KUKA KRL program: draw2.src

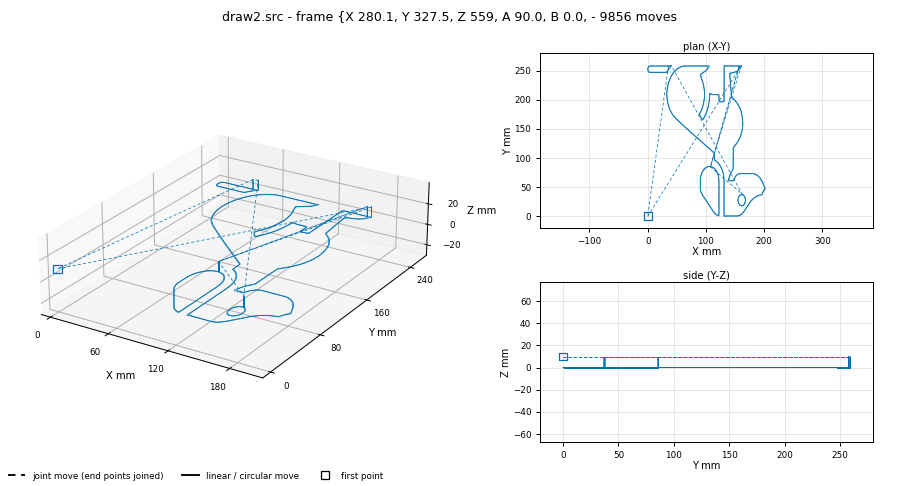
[picture p0: tool path of draw2.src in frame {X 280.1, Y 327.5, Z 559, A 90.0, B 0.0,, 9856 of 9857 moves have a stored position in this frame; points joined in program order, loops and branches not executed]
&ACCESS RVP
&REL 1
DEF DRAW_PICTURE()
; Define home position (pencil up)
POS p_home
p_home = {X 0.00, Y 0.00, Z 10.00, A 0, B 0, C 0}

BAS(#initmov, 0)

$TOOL={X -139.8, Y -0.9, Z 136.2, A 0.0, B 180.0, C 0.0}
$BASE={X 280.1, Y 327.5, Z 559, A 90.0, B 0.0, C 0.0}

PTP $axis_act

PTP p_home

; ----- Contour 1 -----
PTP {X 160.54, Y 258.89, Z 10.00, A 0, B 0, C 0}
LIN {X 160.54, Y 258.89, Z 0.00, A 0, B 0, C 0}
LIN {X 160.34, Y 258.73, Z 0.00, A 0, B 0, C 0} C_DIS
LIN {X 160.14, Y 258.62, Z 0.00, A 0, B 0, C 0} C_DIS
LIN {X 159.93, Y 258.53, Z 0.00, A 0, B 0, C 0} C_DIS
LIN {X 159.72, Y 258.48, Z 0.00, A 0, B 0, C 0} C_DIS
LIN {X 159.50, Y 258.44, Z 0.00, A 0, B 0, C 0} C_DIS
LIN {X 159.29, Y 258.42, Z 0.00, A 0, B 0, C 0} C_DIS
LIN {X 159.07, Y 258.41, Z 0.00, A 0, B 0, C 0} C_DIS
LIN {X 158.85, Y 258.41, Z 0.00, A 0, B 0, C 0} C_DIS
LIN {X 158.63, Y 258.40, Z 0.00, A 0, B 0, C 0} C_DIS
LIN {X 158.41, Y 258.40, Z 0.00, A 0, B 0, C 0} C_DIS
LIN {X 158.20, Y 258.40, Z 0.00, A 0, B 0, C 0} C_DIS
LIN {X 157.98, Y 258.40, Z 0.00, A 0, B 0, C 0} C_DIS
LIN {X 157.76, Y 258.40, Z 0.00, A 0, B 0, C 0} C_DIS
LIN {X 157.54, Y 258.40, Z 0.00, A 0, B 0, C 0} C_DIS
LIN {X 157.33, Y 258.40, Z 0.00, A 0, B 0, C 0} C_DIS
LIN {X 157.11, Y 258.40, Z 0.00, A 0, B 0, C 0} C_DIS
LIN {X 156.89, Y 258.41, Z 0.00, A 0, B 0, C 0} C_DIS
LIN {X 156.67, Y 258.41, Z 0.00, A 0, B 0, C 0} C_DIS
LIN {X 156.46, Y 258.41, Z 0.00, A 0, B 0, C 0} C_DIS
LIN {X 156.24, Y 258.41, Z 0.00, A 0, B 0, C 0} C_DIS
LIN {X 156.02, Y 258.41, Z 0.00, A 0, B 0, C 0} C_DIS
LIN {X 155.81, Y 258.41, Z 0.00, A 0, B 0, C 0} C_DIS
LIN {X 155.59, Y 258.41, Z 0.00, A 0, B 0, C 0} C_DIS
LIN {X 155.37, Y 258.41, Z 0.00, A 0, B 0, C 0} C_DIS
LIN {X 155.15, Y 258.41, Z 0.00, A 0, B 0, C 0} C_DIS
LIN {X 154.94, Y 258.41, Z 0.00, A 0, B 0, C 0} C_DIS
LIN {X 154.72, Y 258.41, Z 0.00, A 0, B 0, C 0} C_DIS
LIN {X 154.50, Y 258.41, Z 0.00, A 0, B 0, C 0} C_DIS
LIN {X 154.28, Y 258.41, Z 0.00, A 0, B 0, C 0} C_DIS
LIN {X 154.07, Y 258.41, Z 0.00, A 0, B 0, C 0} C_DIS
LIN {X 153.85, Y 258.41, Z 0.00, A 0, B 0, C 0} C_DIS
LIN {X 153.63, Y 258.41, Z 0.00, A 0, B 0, C 0} C_DIS
LIN {X 153.41, Y 258.41, Z 0.00, A 0, B 0, C 0} C_DIS
LIN {X 153.20, Y 258.41, Z 0.00, A 0, B 0, C 0} C_DIS
LIN {X 152.98, Y 258.41, Z 0.00, A 0, B 0, C 0} C_DIS
LIN {X 152.76, Y 258.41, Z 0.00, A 0, B 0, C 0} C_DIS
LIN {X 152.54, Y 258.41, Z 0.00, A 0, B 0, C 0} C_DIS
LIN {X 152.33, Y 258.41, Z 0.00, A 0, B 0, C 0} C_DIS
LIN {X 152.11, Y 258.41, Z 0.00, A 0, B 0, C 0} C_DIS
LIN {X 151.89, Y 258.41, Z 0.00, A 0, B 0, C 0} C_DIS
LIN {X 151.67, Y 258.41, Z 0.00, A 0, B 0, C 0} C_DIS
LIN {X 151.46, Y 258.41, Z 0.00, A 0, B 0, C 0} C_DIS
LIN {X 151.24, Y 258.41, Z 0.00, A 0, B 0, C 0} C_DIS
LIN {X 151.02, Y 258.41, Z 0.00, A 0, B 0, C 0} C_DIS
LIN {X 150.80, Y 258.41, Z 0.00, A 0, B 0, C 0} C_DIS
LIN {X 150.59, Y 258.41, Z 0.00, A 0, B 0, C 0} C_DIS
LIN {X 150.37, Y 258.41, Z 0.00, A 0, B 0, C 0} C_DIS
LIN {X 150.15, Y 258.41, Z 0.00, A 0, B 0, C 0} C_DIS
LIN {X 149.93, Y 258.41, Z 0.00, A 0, B 0, C 0} C_DIS
LIN {X 149.72, Y 258.41, Z 0.00, A 0, B 0, C 0} C_DIS
LIN {X 149.50, Y 258.41, Z 0.00, A 0, B 0, C 0} C_DIS
LIN {X 149.28, Y 258.41, Z 0.00, A 0, B 0, C 0} C_DIS
LIN {X 149.06, Y 258.41, Z 0.00, A 0, B 0, C 0} C_DIS
LIN {X 148.85, Y 258.41, Z 0.00, A 0, B 0, C 0} C_DIS
LIN {X 148.63, Y 258.41, Z 0.00, A 0, B 0, C 0} C_DIS
LIN {X 148.41, Y 258.41, Z 0.00, A 0, B 0, C 0} C_DIS
LIN {X 148.19, Y 258.41, Z 0.00, A 0, B 0, C 0} C_DIS
LIN {X 147.98, Y 258.41, Z 0.00, A 0, B 0, C 0} C_DIS
LIN {X 147.76, Y 258.41, Z 0.00, A 0, B 0, C 0} C_DIS
LIN {X 147.54, Y 258.41, Z 0.00, A 0, B 0, C 0} C_DIS
LIN {X 147.33, Y 258.41, Z 0.00, A 0, B 0, C 0} C_DIS
LIN {X 147.11, Y 258.41, Z 0.00, A 0, B 0, C 0} C_DIS
LIN {X 146.89, Y 258.41, Z 0.00, A 0, B 0, C 0} C_DIS
LIN {X 146.67, Y 258.41, Z 0.00, A 0, B 0, C 0} C_DIS
LIN {X 146.46, Y 258.41, Z 0.00, A 0, B 0, C 0} C_DIS
LIN {X 146.24, Y 258.41, Z 0.00, A 0, B 0, C 0} C_DIS
LIN {X 146.02, Y 258.41, Z 0.00, A 0, B 0, C 0} C_DIS
LIN {X 145.80, Y 258.41, Z 0.00, A 0, B 0, C 0} C_DIS
LIN {X 145.59, Y 258.41, Z 0.00, A 0, B 0, C 0} C_DIS
LIN {X 145.37, Y 258.41, Z 0.00, A 0, B 0, C 0} C_DIS
LIN {X 145.15, Y 258.41, Z 0.00, A 0, B 0, C 0} C_DIS
LIN {X 144.93, Y 258.41, Z 0.00, A 0, B 0, C 0} C_DIS
LIN {X 144.72, Y 258.41, Z 0.00, A 0, B 0, C 0} C_DIS
LIN {X 144.50, Y 258.41, Z 0.00, A 0, B 0, C 0} C_DIS
LIN {X 144.28, Y 258.41, Z 0.00, A 0, B 0, C 0} C_DIS
LIN {X 144.06, Y 258.41, Z 0.00, A 0, B 0, C 0} C_DIS
LIN {X 143.85, Y 258.41, Z 0.00, A 0, B 0, C 0} C_DIS
LIN {X 143.63, Y 258.41, Z 0.00, A 0, B 0, C 0} C_DIS
LIN {X 143.41, Y 258.41, Z 0.00, A 0, B 0, C 0} C_DIS
LIN {X 143.19, Y 258.41, Z 0.00, A 0, B 0, C 0} C_DIS
LIN {X 142.98, Y 258.41, Z 0.00, A 0, B 0, C 0} C_DIS
LIN {X 142.76, Y 258.41, Z 0.00, A 0, B 0, C 0} C_DIS
LIN {X 142.54, Y 258.41, Z 0.00, A 0, B 0, C 0} C_DIS
LIN {X 142.32, Y 258.41, Z 0.00, A 0, B 0, C 0} C_DIS
LIN {X 142.11, Y 258.41, Z 0.00, A 0, B 0, C 0} C_DIS
LIN {X 141.89, Y 258.41, Z 0.00, A 0, B 0, C 0} C_DIS
LIN {X 141.67, Y 258.41, Z 0.00, A 0, B 0, C 0} C_DIS
LIN {X 141.45, Y 258.41, Z 0.00, A 0, B 0, C 0} C_DIS
LIN {X 141.24, Y 258.41, Z 0.00, A 0, B 0, C 0} C_DIS
LIN {X 141.02, Y 258.41, Z 0.00, A 0, B 0, C 0} C_DIS
LIN {X 140.80, Y 258.41, Z 0.00, A 0, B 0, C 0} C_DIS
LIN {X 140.58, Y 258.41, Z 0.00, A 0, B 0, C 0} C_DIS
LIN {X 140.37, Y 258.41, Z 0.00, A 0, B 0, C 0} C_DIS
LIN {X 140.15, Y 258.41, Z 0.00, A 0, B 0, C 0} C_DIS
LIN {X 139.93, Y 258.41, Z 0.00, A 0, B 0, C 0} C_DIS
LIN {X 139.71, Y 258.41, Z 0.00, A 0, B 0, C 0} C_DIS
LIN {X 139.50, Y 258.41, Z 0.00, A 0, B 0, C 0} C_DIS
LIN {X 139.28, Y 258.41, Z 0.00, A 0, B 0, C 0} C_DIS
LIN {X 139.06, Y 258.41, Z 0.00, A 0, B 0, C 0} C_DIS
LIN {X 138.85, Y 258.41, Z 0.00, A 0, B 0, C 0} C_DIS
LIN {X 138.63, Y 258.41, Z 0.00, A 0, B 0, C 0} C_DIS
LIN {X 138.41, Y 258.41, Z 0.00, A 0, B 0, C 0} C_DIS
LIN {X 138.19, Y 258.41, Z 0.00, A 0, B 0, C 0} C_DIS
LIN {X 137.98, Y 258.41, Z 0.00, A 0, B 0, C 0} C_DIS
LIN {X 137.76, Y 258.41, Z 0.00, A 0, B 0, C 0} C_DIS
LIN {X 137.54, Y 258.40, Z 0.00, A 0, B 0, C 0} C_DIS
LIN {X 137.32, Y 258.40, Z 0.00, A 0, B 0, C 0} C_DIS
LIN {X 137.11, Y 258.40, Z 0.00, A 0, B 0, C 0} C_DIS
LIN {X 136.89, Y 258.40, Z 0.00, A 0, B 0, C 0} C_DIS
LIN {X 136.67, Y 258.40, Z 0.00, A 0, B 0, C 0} C_DIS
LIN {X 136.45, Y 258.40, Z 0.00, A 0, B 0, C 0} C_DIS
LIN {X 136.24, Y 258.40, Z 0.00, A 0, B 0, C 0} C_DIS
LIN {X 136.02, Y 258.40, Z 0.00, A 0, B 0, C 0} C_DIS
LIN {X 135.80, Y 258.41, Z 0.00, A 0, B 0, C 0} C_DIS
LIN {X 135.58, Y 258.41, Z 0.00, A 0, B 0, C 0} C_DIS
LIN {X 135.37, Y 258.41, Z 0.00, A 0, B 0, C 0} C_DIS
LIN {X 135.15, Y 258.41, Z 0.00, A 0, B 0, C 0} C_DIS
LIN {X 134.93, Y 258.41, Z 0.00, A 0, B 0, C 0} C_DIS
LIN {X 134.72, Y 258.41, Z 0.00, A 0, B 0, C 0} C_DIS
LIN {X 134.50, Y 258.41, Z 0.00, A 0, B 0, C 0} C_DIS
LIN {X 134.28, Y 258.41, Z 0.00, A 0, B 0, C 0} C_DIS
LIN {X 134.06, Y 258.41, Z 0.00, A 0, B 0, C 0} C_DIS
LIN {X 133.84, Y 258.41, Z 0.00, A 0, B 0, C 0} C_DIS
LIN {X 133.63, Y 258.40, Z 0.00, A 0, B 0, C 0} C_DIS
LIN {X 133.41, Y 258.40, Z 0.00, A 0, B 0, C 0} C_DIS
LIN {X 133.19, Y 258.39, Z 0.00, A 0, B 0, C 0} C_DIS
LIN {X 132.97, Y 258.39, Z 0.00, A 0, B 0, C 0} C_DIS
LIN {X 132.75, Y 258.39, Z 0.00, A 0, B 0, C 0} C_DIS
LIN {X 132.54, Y 258.41, Z 0.00, A 0, B 0, C 0} C_DIS
LIN {X 132.32, Y 258.43, Z 0.00, A 0, B 0, C 0} C_DIS
LIN {X 132.11, Y 258.47, Z 0.00, A 0, B 0, C 0} C_DIS
LIN {X 131.90, Y 258.53, Z 0.00, A 0, B 0, C 0} C_DIS
LIN {X 131.69, Y 258.59, Z 0.00, A 0, B 0, C 0} C_DIS
LIN {X 131.47, Y 258.66, Z 0.00, A 0, B 0, C 0} C_DIS
LIN {X 131.25, Y 258.71, Z 0.00, A 0, B 0, C 0} C_DIS
LIN {X 131.03, Y 258.70, Z 0.00, A 0, B 0, C 0} C_DIS
LIN {X 130.84, Y 258.58, Z 0.00, A 0, B 0, C 0} C_DIS
LIN {X 130.73, Y 258.32, Z 0.00, A 0, B 0, C 0} C_DIS
LIN {X 130.70, Y 257.99, Z 0.00, A 0, B 0, C 0} C_DIS
LIN {X 130.73, Y 257.65, Z 0.00, A 0, B 0, C 0} C_DIS
LIN {X 130.77, Y 257.33, Z 0.00, A 0, B 0, C 0} C_DIS
LIN {X 130.83, Y 257.01, Z 0.00, A 0, B 0, C 0} C_DIS
LIN {X 130.87, Y 256.70, Z 0.00, A 0, B 0, C 0} C_DIS
LIN {X 130.90, Y 256.37, Z 0.00, A 0, B 0, C 0} C_DIS
LIN {X 130.91, Y 256.05, Z 0.00, A 0, B 0, C 0} C_DIS
LIN {X 130.91, Y 255.72, Z 0.00, A 0, B 0, C 0} C_DIS
LIN {X 130.91, Y 255.39, Z 0.00, A 0, B 0, C 0} C_DIS
LIN {X 130.91, Y 255.06, Z 0.00, A 0, B 0, C 0} C_DIS
LIN {X 130.91, Y 254.73, Z 0.00, A 0, B 0, C 0} C_DIS
LIN {X 130.91, Y 254.40, Z 0.00, A 0, B 0, C 0} C_DIS
LIN {X 130.91, Y 254.08, Z 0.00, A 0, B 0, C 0} C_DIS
LIN {X 130.91, Y 253.75, Z 0.00, A 0, B 0, C 0} C_DIS
LIN {X 130.91, Y 253.42, Z 0.00, A 0, B 0, C 0} C_DIS
LIN {X 130.91, Y 253.10, Z 0.00, A 0, B 0, C 0} C_DIS
LIN {X 130.91, Y 252.77, Z 0.00, A 0, B 0, C 0} C_DIS
LIN {X 130.91, Y 252.44, Z 0.00, A 0, B 0, C 0} C_DIS
LIN {X 130.91, Y 252.11, Z 0.00, A 0, B 0, C 0} C_DIS
LIN {X 130.91, Y 251.78, Z 0.00, A 0, B 0, C 0} C_DIS
LIN {X 130.91, Y 251.46, Z 0.00, A 0, B 0, C 0} C_DIS
LIN {X 130.91, Y 251.13, Z 0.00, A 0, B 0, C 0} C_DIS
LIN {X 130.91, Y 250.80, Z 0.00, A 0, B 0, C 0} C_DIS
LIN {X 130.91, Y 250.47, Z 0.00, A 0, B 0, C 0} C_DIS
LIN {X 130.91, Y 250.15, Z 0.00, A 0, B 0, C 0} C_DIS
LIN {X 130.91, Y 249.82, Z 0.00, A 0, B 0, C 0} C_DIS
LIN {X 130.91, Y 249.49, Z 0.00, A 0, B 0, C 0} C_DIS
LIN {X 130.91, Y 249.16, Z 0.00, A 0, B 0, C 0} C_DIS
LIN {X 130.91, Y 248.84, Z 0.00, A 0, B 0, C 0} C_DIS
LIN {X 130.91, Y 248.51, Z 0.00, A 0, B 0, C 0} C_DIS
LIN {X 130.91, Y 248.18, Z 0.00, A 0, B 0, C 0} C_DIS
LIN {X 130.91, Y 247.85, Z 0.00, A 0, B 0, C 0} C_DIS
LIN {X 130.91, Y 247.52, Z 0.00, A 0, B 0, C 0} C_DIS
LIN {X 130.91, Y 247.20, Z 0.00, A 0, B 0, C 0} C_DIS
LIN {X 130.91, Y 246.87, Z 0.00, A 0, B 0, C 0} C_DIS
LIN {X 130.91, Y 246.54, Z 0.00, A 0, B 0, C 0} C_DIS
LIN {X 130.91, Y 246.21, Z 0.00, A 0, B 0, C 0} C_DIS
LIN {X 130.91, Y 245.89, Z 0.00, A 0, B 0, C 0} C_DIS
LIN {X 130.91, Y 245.56, Z 0.00, A 0, B 0, C 0} C_DIS
LIN {X 130.91, Y 245.23, Z 0.00, A 0, B 0, C 0} C_DIS
LIN {X 130.91, Y 244.90, Z 0.00, A 0, B 0, C 0} C_DIS
LIN {X 130.91, Y 244.58, Z 0.00, A 0, B 0, C 0} C_DIS
LIN {X 130.91, Y 244.25, Z 0.00, A 0, B 0, C 0} C_DIS
LIN {X 130.91, Y 243.92, Z 0.00, A 0, B 0, C 0} C_DIS
LIN {X 130.91, Y 243.59, Z 0.00, A 0, B 0, C 0} C_DIS
LIN {X 130.91, Y 243.26, Z 0.00, A 0, B 0, C 0} C_DIS
LIN {X 130.91, Y 242.94, Z 0.00, A 0, B 0, C 0} C_DIS
LIN {X 130.91, Y 242.61, Z 0.00, A 0, B 0, C 0} C_DIS
LIN {X 130.91, Y 242.28, Z 0.00, A 0, B 0, C 0} C_DIS
LIN {X 130.91, Y 241.95, Z 0.00, A 0, B 0, C 0} C_DIS
LIN {X 130.91, Y 241.63, Z 0.00, A 0, B 0, C 0} C_DIS
LIN {X 130.91, Y 241.30, Z 0.00, A 0, B 0, C 0} C_DIS
LIN {X 130.91, Y 240.97, Z 0.00, A 0, B 0, C 0} C_DIS
LIN {X 130.91, Y 240.64, Z 0.00, A 0, B 0, C 0} C_DIS
LIN {X 130.91, Y 240.32, Z 0.00, A 0, B 0, C 0} C_DIS
LIN {X 130.91, Y 239.99, Z 0.00, A 0, B 0, C 0} C_DIS
LIN {X 130.91, Y 239.66, Z 0.00, A 0, B 0, C 0} C_DIS
LIN {X 130.91, Y 239.33, Z 0.00, A 0, B 0, C 0} C_DIS
LIN {X 130.91, Y 239.00, Z 0.00, A 0, B 0, C 0} C_DIS
LIN {X 130.91, Y 238.68, Z 0.00, A 0, B 0, C 0} C_DIS
LIN {X 130.91, Y 238.35, Z 0.00, A 0, B 0, C 0} C_DIS
LIN {X 130.91, Y 238.02, Z 0.00, A 0, B 0, C 0} C_DIS
LIN {X 130.91, Y 237.69, Z 0.00, A 0, B 0, C 0} C_DIS
LIN {X 130.91, Y 237.37, Z 0.00, A 0, B 0, C 0} C_DIS
LIN {X 130.91, Y 237.04, Z 0.00, A 0, B 0, C 0} C_DIS
LIN {X 130.91, Y 236.71, Z 0.00, A 0, B 0, C 0} C_DIS
LIN {X 130.91, Y 236.38, Z 0.00, A 0, B 0, C 0} C_DIS
LIN {X 130.91, Y 236.06, Z 0.00, A 0, B 0, C 0} C_DIS
LIN {X 130.91, Y 235.73, Z 0.00, A 0, B 0, C 0} C_DIS
LIN {X 130.91, Y 235.40, Z 0.00, A 0, B 0, C 0} C_DIS
LIN {X 130.91, Y 235.07, Z 0.00, A 0, B 0, C 0} C_DIS
LIN {X 130.91, Y 234.74, Z 0.00, A 0, B 0, C 0} C_DIS
LIN {X 130.91, Y 234.42, Z 0.00, A 0, B 0, C 0} C_DIS
LIN {X 130.91, Y 234.09, Z 0.00, A 0, B 0, C 0} C_DIS
LIN {X 130.91, Y 233.76, Z 0.00, A 0, B 0, C 0} C_DIS
LIN {X 130.91, Y 233.43, Z 0.00, A 0, B 0, C 0} C_DIS
LIN {X 130.91, Y 233.11, Z 0.00, A 0, B 0, C 0} C_DIS
LIN {X 130.91, Y 232.78, Z 0.00, A 0, B 0, C 0} C_DIS
LIN {X 130.91, Y 232.45, Z 0.00, A 0, B 0, C 0} C_DIS
LIN {X 130.91, Y 232.12, Z 0.00, A 0, B 0, C 0} C_DIS
LIN {X 130.91, Y 231.80, Z 0.00, A 0, B 0, C 0} C_DIS
LIN {X 130.91, Y 231.47, Z 0.00, A 0, B 0, C 0} C_DIS
LIN {X 130.91, Y 231.14, Z 0.00, A 0, B 0, C 0} C_DIS
LIN {X 130.91, Y 230.81, Z 0.00, A 0, B 0, C 0} C_DIS
LIN {X 130.91, Y 230.48, Z 0.00, A 0, B 0, C 0} C_DIS
LIN {X 130.91, Y 230.16, Z 0.00, A 0, B 0, C 0} C_DIS
LIN {X 130.91, Y 229.83, Z 0.00, A 0, B 0, C 0} C_DIS
LIN {X 130.91, Y 229.50, Z 0.00, A 0, B 0, C 0} C_DIS
LIN {X 130.91, Y 229.17, Z 0.00, A 0, B 0, C 0} C_DIS
LIN {X 130.91, Y 228.85, Z 0.00, A 0, B 0, C 0} C_DIS
LIN {X 130.91, Y 228.52, Z 0.00, A 0, B 0, C 0} C_DIS
LIN {X 130.91, Y 228.19, Z 0.00, A 0, B 0, C 0} C_DIS
LIN {X 130.91, Y 227.86, Z 0.00, A 0, B 0, C 0} C_DIS
LIN {X 130.91, Y 227.54, Z 0.00, A 0, B 0, C 0} C_DIS
LIN {X 130.91, Y 227.21, Z 0.00, A 0, B 0, C 0} C_DIS
LIN {X 130.91, Y 226.88, Z 0.00, A 0, B 0, C 0} C_DIS
LIN {X 130.91, Y 226.55, Z 0.00, A 0, B 0, C 0} C_DIS
LIN {X 130.91, Y 226.22, Z 0.00, A 0, B 0, C 0} C_DIS
LIN {X 130.91, Y 225.90, Z 0.00, A 0, B 0, C 0} C_DIS
LIN {X 130.91, Y 225.57, Z 0.00, A 0, B 0, C 0} C_DIS
LIN {X 130.91, Y 225.24, Z 0.00, A 0, B 0, C 0} C_DIS
LIN {X 130.91, Y 224.91, Z 0.00, A 0, B 0, C 0} C_DIS
LIN {X 130.91, Y 224.59, Z 0.00, A 0, B 0, C 0} C_DIS
LIN {X 130.91, Y 224.26, Z 0.00, A 0, B 0, C 0} C_DIS
LIN {X 130.91, Y 223.93, Z 0.00, A 0, B 0, C 0} C_DIS
LIN {X 130.91, Y 223.60, Z 0.00, A 0, B 0, C 0} C_DIS
LIN {X 130.91, Y 223.28, Z 0.00, A 0, B 0, C 0} C_DIS
LIN {X 130.91, Y 222.95, Z 0.00, A 0, B 0, C 0} C_DIS
LIN {X 130.91, Y 222.62, Z 0.00, A 0, B 0, C 0} C_DIS
LIN {X 130.91, Y 222.29, Z 0.00, A 0, B 0, C 0} C_DIS
LIN {X 130.91, Y 221.96, Z 0.00, A 0, B 0, C 0} C_DIS
LIN {X 130.91, Y 221.64, Z 0.00, A 0, B 0, C 0} C_DIS
LIN {X 130.91, Y 221.31, Z 0.00, A 0, B 0, C 0} C_DIS
LIN {X 130.91, Y 220.98, Z 0.00, A 0, B 0, C 0} C_DIS
LIN {X 130.91, Y 220.65, Z 0.00, A 0, B 0, C 0} C_DIS
LIN {X 130.91, Y 220.33, Z 0.00, A 0, B 0, C 0} C_DIS
LIN {X 130.91, Y 220.00, Z 0.00, A 0, B 0, C 0} C_DIS
LIN {X 130.91, Y 219.67, Z 0.00, A 0, B 0, C 0} C_DIS
LIN {X 130.91, Y 219.34, Z 0.00, A 0, B 0, C 0} C_DIS
LIN {X 130.91, Y 219.02, Z 0.00, A 0, B 0, C 0} C_DIS
LIN {X 130.91, Y 218.69, Z 0.00, A 0, B 0, C 0} C_DIS
LIN {X 130.91, Y 218.36, Z 0.00, A 0, B 0, C 0} C_DIS
LIN {X 130.91, Y 218.03, Z 0.00, A 0, B 0, C 0} C_DIS
LIN {X 130.91, Y 217.70, Z 0.00, A 0, B 0, C 0} C_DIS
LIN {X 130.91, Y 217.38, Z 0.00, A 0, B 0, C 0} C_DIS
LIN {X 130.91, Y 217.05, Z 0.00, A 0, B 0, C 0} C_DIS
LIN {X 130.91, Y 216.72, Z 0.00, A 0, B 0, C 0} C_DIS
LIN {X 130.91, Y 216.39, Z 0.00, A 0, B 0, C 0} C_DIS
LIN {X 130.91, Y 216.07, Z 0.00, A 0, B 0, C 0} C_DIS
LIN {X 130.91, Y 215.74, Z 0.00, A 0, B 0, C 0} C_DIS
LIN {X 130.91, Y 215.41, Z 0.00, A 0, B 0, C 0} C_DIS
LIN {X 130.91, Y 215.08, Z 0.00, A 0, B 0, C 0} C_DIS
LIN {X 130.91, Y 214.76, Z 0.00, A 0, B 0, C 0} C_DIS
LIN {X 130.91, Y 214.43, Z 0.00, A 0, B 0, C 0} C_DIS
LIN {X 130.91, Y 214.10, Z 0.00, A 0, B 0, C 0} C_DIS
LIN {X 130.91, Y 213.77, Z 0.00, A 0, B 0, C 0} C_DIS
LIN {X 130.91, Y 213.44, Z 0.00, A 0, B 0, C 0} C_DIS
LIN {X 130.91, Y 213.12, Z 0.00, A 0, B 0, C 0} C_DIS
LIN {X 130.91, Y 212.79, Z 0.00, A 0, B 0, C 0} C_DIS
LIN {X 130.91, Y 212.46, Z 0.00, A 0, B 0, C 0} C_DIS
LIN {X 130.91, Y 212.13, Z 0.00, A 0, B 0, C 0} C_DIS
LIN {X 130.91, Y 211.81, Z 0.00, A 0, B 0, C 0} C_DIS
LIN {X 130.91, Y 211.48, Z 0.00, A 0, B 0, C 0} C_DIS
LIN {X 130.91, Y 211.15, Z 0.00, A 0, B 0, C 0} C_DIS
LIN {X 130.91, Y 210.82, Z 0.00, A 0, B 0, C 0} C_DIS
LIN {X 130.91, Y 210.50, Z 0.00, A 0, B 0, C 0} C_DIS
LIN {X 130.91, Y 210.17, Z 0.00, A 0, B 0, C 0} C_DIS
LIN {X 130.91, Y 209.84, Z 0.00, A 0, B 0, C 0} C_DIS
LIN {X 130.91, Y 209.51, Z 0.00, A 0, B 0, C 0} C_DIS
LIN {X 130.91, Y 209.18, Z 0.00, A 0, B 0, C 0} C_DIS
LIN {X 130.91, Y 208.86, Z 0.00, A 0, B 0, C 0} C_DIS
LIN {X 130.91, Y 208.53, Z 0.00, A 0, B 0, C 0} C_DIS
LIN {X 130.91, Y 208.20, Z 0.00, A 0, B 0, C 0} C_DIS
LIN {X 130.91, Y 207.87, Z 0.00, A 0, B 0, C 0} C_DIS
LIN {X 130.91, Y 207.55, Z 0.00, A 0, B 0, C 0} C_DIS
LIN {X 130.91, Y 207.22, Z 0.00, A 0, B 0, C 0} C_DIS
LIN {X 130.91, Y 206.89, Z 0.00, A 0, B 0, C 0} C_DIS
LIN {X 130.91, Y 206.56, Z 0.00, A 0, B 0, C 0} C_DIS
LIN {X 130.91, Y 206.24, Z 0.00, A 0, B 0, C 0} C_DIS
LIN {X 130.91, Y 205.91, Z 0.00, A 0, B 0, C 0} C_DIS
LIN {X 130.91, Y 205.58, Z 0.00, A 0, B 0, C 0} C_DIS
LIN {X 130.91, Y 205.25, Z 0.00, A 0, B 0, C 0} C_DIS
LIN {X 130.91, Y 204.92, Z 0.00, A 0, B 0, C 0} C_DIS
LIN {X 130.91, Y 204.60, Z 0.00, A 0, B 0, C 0} C_DIS
LIN {X 130.91, Y 204.27, Z 0.00, A 0, B 0, C 0} C_DIS
LIN {X 130.91, Y 203.94, Z 0.00, A 0, B 0, C 0} C_DIS
LIN {X 130.91, Y 203.61, Z 0.00, A 0, B 0, C 0} C_DIS
LIN {X 130.91, Y 203.29, Z 0.00, A 0, B 0, C 0} C_DIS
LIN {X 130.92, Y 202.96, Z 0.00, A 0, B 0, C 0} C_DIS
LIN {X 130.92, Y 202.63, Z 0.00, A 0, B 0, C 0} C_DIS
LIN {X 130.92, Y 202.30, Z 0.00, A 0, B 0, C 0} C_DIS
LIN {X 130.92, Y 201.98, Z 0.00, A 0, B 0, C 0} C_DIS
LIN {X 130.92, Y 201.65, Z 0.00, A 0, B 0, C 0} C_DIS
LIN {X 130.91, Y 201.32, Z 0.00, A 0, B 0, C 0} C_DIS
LIN {X 130.91, Y 200.99, Z 0.00, A 0, B 0, C 0} C_DIS
LIN {X 130.91, Y 200.67, Z 0.00, A 0, B 0, C 0} C_DIS
LIN {X 130.90, Y 200.34, Z 0.00, A 0, B 0, C 0} C_DIS
LIN {X 130.88, Y 200.01, Z 0.00, A 0, B 0, C 0} C_DIS
LIN {X 130.84, Y 199.69, Z 0.00, A 0, B 0, C 0} C_DIS
LIN {X 130.78, Y 199.38, Z 0.00, A 0, B 0, C 0} C_DIS
LIN {X 130.73, Y 199.05, Z 0.00, A 0, B 0, C 0} C_DIS
LIN {X 130.67, Y 198.74, Z 0.00, A 0, B 0, C 0} C_DIS
LIN {X 130.58, Y 198.44, Z 0.00, A 0, B 0, C 0} C_DIS
LIN {X 130.45, Y 198.19, Z 0.00, A 0, B 0, C 0} C_DIS
LIN {X 130.30, Y 197.95, Z 0.00, A 0, B 0, C 0} C_DIS
LIN {X 130.14, Y 197.71, Z 0.00, A 0, B 0, C 0} C_DIS
LIN {X 129.98, Y 197.49, Z 0.00, A 0, B 0, C 0} C_DIS
LIN {X 129.81, Y 197.30, Z 0.00, A 0, B 0, C 0} C_DIS
LIN {X 129.62, Y 197.16, Z 0.00, A 0, B 0, C 0} C_DIS
LIN {X 129.42, Y 197.05, Z 0.00, A 0, B 0, C 0} C_DIS
LIN {X 129.20, Y 196.98, Z 0.00, A 0, B 0, C 0} C_DIS
LIN {X 128.98, Y 196.91, Z 0.00, A 0, B 0, C 0} C_DIS
LIN {X 128.77, Y 196.86, Z 0.00, A 0, B 0, C 0} C_DIS
LIN {X 128.56, Y 196.82, Z 0.00, A 0, B 0, C 0} C_DIS
LIN {X 128.34, Y 196.80, Z 0.00, A 0, B 0, C 0} C_DIS
LIN {X 128.12, Y 196.78, Z 0.00, A 0, B 0, C 0} C_DIS
LIN {X 127.91, Y 196.78, Z 0.00, A 0, B 0, C 0} C_DIS
LIN {X 127.69, Y 196.78, Z 0.00, A 0, B 0, C 0} C_DIS
LIN {X 127.47, Y 196.79, Z 0.00, A 0, B 0, C 0} C_DIS
LIN {X 127.26, Y 196.79, Z 0.00, A 0, B 0, C 0} C_DIS
LIN {X 127.04, Y 196.80, Z 0.00, A 0, B 0, C 0} C_DIS
LIN {X 126.82, Y 196.81, Z 0.00, A 0, B 0, C 0} C_DIS
LIN {X 126.60, Y 196.81, Z 0.00, A 0, B 0, C 0} C_DIS
LIN {X 126.38, Y 196.80, Z 0.00, A 0, B 0, C 0} C_DIS
LIN {X 126.17, Y 196.79, Z 0.00, A 0, B 0, C 0} C_DIS
LIN {X 125.95, Y 196.79, Z 0.00, A 0, B 0, C 0} C_DIS
LIN {X 125.73, Y 196.78, Z 0.00, A 0, B 0, C 0} C_DIS
LIN {X 125.51, Y 196.78, Z 0.00, A 0, B 0, C 0} C_DIS
LIN {X 125.30, Y 196.79, Z 0.00, A 0, B 0, C 0} C_DIS
LIN {X 125.08, Y 196.80, Z 0.00, A 0, B 0, C 0} C_DIS
LIN {X 124.86, Y 196.83, Z 0.00, A 0, B 0, C 0} C_DIS
LIN {X 124.65, Y 196.87, Z 0.00, A 0, B 0, C 0} C_DIS
LIN {X 124.43, Y 196.92, Z 0.00, A 0, B 0, C 0} C_DIS
LIN {X 124.22, Y 197.00, Z 0.00, A 0, B 0, C 0} C_DIS
LIN {X 124.01, Y 197.09, Z 0.00, A 0, B 0, C 0} C_DIS
LIN {X 123.80, Y 197.19, Z 0.00, A 0, B 0, C 0} C_DIS
LIN {X 123.61, Y 197.33, Z 0.00, A 0, B 0, C 0} C_DIS
LIN {X 123.45, Y 197.54, Z 0.00, A 0, B 0, C 0} C_DIS
LIN {X 123.30, Y 197.78, Z 0.00, A 0, B 0, C 0} C_DIS
LIN {X 123.14, Y 198.01, Z 0.00, A 0, B 0, C 0} C_DIS
LIN {X 122.99, Y 198.24, Z 0.00, A 0, B 0, C 0} C_DIS
LIN {X 122.87, Y 198.51, Z 0.00, A 0, B 0, C 0} C_DIS
LIN {X 122.79, Y 198.82, Z 0.00, A 0, B 0, C 0} C_DIS
LIN {X 122.73, Y 199.13, Z 0.00, A 0, B 0, C 0} C_DIS
LIN {X 122.67, Y 199.45, Z 0.00, A 0, B 0, C 0} C_DIS
LIN {X 122.63, Y 199.77, Z 0.00, A 0, B 0, C 0} C_DIS
LIN {X 122.60, Y 200.10, Z 0.00, A 0, B 0, C 0} C_DIS
LIN {X 122.58, Y 200.42, Z 0.00, A 0, B 0, C 0} C_DIS
LIN {X 122.56, Y 200.75, Z 0.00, A 0, B 0, C 0} C_DIS
LIN {X 122.56, Y 201.07, Z 0.00, A 0, B 0, C 0} C_DIS
LIN {X 122.55, Y 201.40, Z 0.00, A 0, B 0, C 0} C_DIS
LIN {X 122.55, Y 201.73, Z 0.00, A 0, B 0, C 0} C_DIS
LIN {X 122.56, Y 202.06, Z 0.00, A 0, B 0, C 0} C_DIS
LIN {X 122.56, Y 202.39, Z 0.00, A 0, B 0, C 0} C_DIS
LIN {X 122.56, Y 202.71, Z 0.00, A 0, B 0, C 0} C_DIS
LIN {X 122.57, Y 203.04, Z 0.00, A 0, B 0, C 0} C_DIS
LIN {X 122.57, Y 203.37, Z 0.00, A 0, B 0, C 0} C_DIS
LIN {X 122.57, Y 203.70, Z 0.00, A 0, B 0, C 0} C_DIS
LIN {X 122.57, Y 204.02, Z 0.00, A 0, B 0, C 0} C_DIS
LIN {X 122.57, Y 204.35, Z 0.00, A 0, B 0, C 0} C_DIS
LIN {X 122.56, Y 204.68, Z 0.00, A 0, B 0, C 0} C_DIS
LIN {X 122.56, Y 205.01, Z 0.00, A 0, B 0, C 0} C_DIS
LIN {X 122.56, Y 205.33, Z 0.00, A 0, B 0, C 0} C_DIS
LIN {X 122.56, Y 205.66, Z 0.00, A 0, B 0, C 0} C_DIS
LIN {X 122.56, Y 205.99, Z 0.00, A 0, B 0, C 0} C_DIS
LIN {X 122.55, Y 206.32, Z 0.00, A 0, B 0, C 0} C_DIS
LIN {X 122.56, Y 206.65, Z 0.00, A 0, B 0, C 0} C_DIS
LIN {X 122.56, Y 206.97, Z 0.00, A 0, B 0, C 0} C_DIS
LIN {X 122.57, Y 207.30, Z 0.00, A 0, B 0, C 0} C_DIS
LIN {X 122.58, Y 207.63, Z 0.00, A 0, B 0, C 0} C_DIS
LIN {X 122.56, Y 207.95, Z 0.00, A 0, B 0, C 0} C_DIS
LIN {X 122.52, Y 208.28, Z 0.00, A 0, B 0, C 0} C_DIS
LIN {X 122.43, Y 208.59, Z 0.00, A 0, B 0, C 0} C_DIS
LIN {X 122.31, Y 208.87, Z 0.00, A 0, B 0, C 0} C_DIS
LIN {X 122.15, Y 209.07, Z 0.00, A 0, B 0, C 0} C_DIS
LIN {X 121.95, Y 209.17, Z 0.00, A 0, B 0, C 0} C_DIS
LIN {X 121.74, Y 209.22, Z 0.00, A 0, B 0, C 0} C_DIS
LIN {X 121.52, Y 209.24, Z 0.00, A 0, B 0, C 0} C_DIS
LIN {X 121.30, Y 209.24, Z 0.00, A 0, B 0, C 0} C_DIS
LIN {X 121.08, Y 209.25, Z 0.00, A 0, B 0, C 0} C_DIS
LIN {X 120.86, Y 209.25, Z 0.00, A 0, B 0, C 0} C_DIS
LIN {X 120.64, Y 209.25, Z 0.00, A 0, B 0, C 0} C_DIS
LIN {X 120.42, Y 209.25, Z 0.00, A 0, B 0, C 0} C_DIS
LIN {X 120.20, Y 209.25, Z 0.00, A 0, B 0, C 0} C_DIS
LIN {X 119.99, Y 209.25, Z 0.00, A 0, B 0, C 0} C_DIS
LIN {X 119.77, Y 209.25, Z 0.00, A 0, B 0, C 0} C_DIS
LIN {X 119.56, Y 209.25, Z 0.00, A 0, B 0, C 0} C_DIS
LIN {X 119.34, Y 209.25, Z 0.00, A 0, B 0, C 0} C_DIS
LIN {X 119.12, Y 209.25, Z 0.00, A 0, B 0, C 0} C_DIS
LIN {X 118.91, Y 209.25, Z 0.00, A 0, B 0, C 0} C_DIS
LIN {X 118.69, Y 209.25, Z 0.00, A 0, B 0, C 0} C_DIS
LIN {X 118.47, Y 209.25, Z 0.00, A 0, B 0, C 0} C_DIS
LIN {X 118.25, Y 209.25, Z 0.00, A 0, B 0, C 0} C_DIS
LIN {X 118.04, Y 209.24, Z 0.00, A 0, B 0, C 0} C_DIS
LIN {X 117.82, Y 209.24, Z 0.00, A 0, B 0, C 0} C_DIS
LIN {X 117.60, Y 209.24, Z 0.00, A 0, B 0, C 0} C_DIS
LIN {X 117.38, Y 209.24, Z 0.00, A 0, B 0, C 0} C_DIS
LIN {X 117.16, Y 209.24, Z 0.00, A 0, B 0, C 0} C_DIS
LIN {X 116.95, Y 209.24, Z 0.00, A 0, B 0, C 0} C_DIS
LIN {X 116.73, Y 209.24, Z 0.00, A 0, B 0, C 0} C_DIS
LIN {X 116.51, Y 209.24, Z 0.00, A 0, B 0, C 0} C_DIS
LIN {X 116.29, Y 209.25, Z 0.00, A 0, B 0, C 0} C_DIS
LIN {X 116.08, Y 209.25, Z 0.00, A 0, B 0, C 0} C_DIS
LIN {X 115.86, Y 209.25, Z 0.00, A 0, B 0, C 0} C_DIS
LIN {X 115.64, Y 209.25, Z 0.00, A 0, B 0, C 0} C_DIS
LIN {X 115.42, Y 209.25, Z 0.00, A 0, B 0, C 0} C_DIS
LIN {X 115.21, Y 209.25, Z 0.00, A 0, B 0, C 0} C_DIS
LIN {X 114.99, Y 209.26, Z 0.00, A 0, B 0, C 0} C_DIS
LIN {X 114.77, Y 209.26, Z 0.00, A 0, B 0, C 0} C_DIS
LIN {X 114.56, Y 209.26, Z 0.00, A 0, B 0, C 0} C_DIS
LIN {X 114.34, Y 209.26, Z 0.00, A 0, B 0, C 0} C_DIS
LIN {X 114.12, Y 209.25, Z 0.00, A 0, B 0, C 0} C_DIS
LIN {X 113.90, Y 209.25, Z 0.00, A 0, B 0, C 0} C_DIS
LIN {X 113.69, Y 209.24, Z 0.00, A 0, B 0, C 0} C_DIS
LIN {X 113.47, Y 209.24, Z 0.00, A 0, B 0, C 0} C_DIS
LIN {X 113.25, Y 209.23, Z 0.00, A 0, B 0, C 0} C_DIS
LIN {X 113.03, Y 209.23, Z 0.00, A 0, B 0, C 0} C_DIS
LIN {X 112.81, Y 209.23, Z 0.00, A 0, B 0, C 0} C_DIS
LIN {X 112.60, Y 209.24, Z 0.00, A 0, B 0, C 0} C_DIS
LIN {X 112.38, Y 209.26, Z 0.00, A 0, B 0, C 0} C_DIS
LIN {X 112.16, Y 209.30, Z 0.00, A 0, B 0, C 0} C_DIS
LIN {X 111.95, Y 209.35, Z 0.00, A 0, B 0, C 0} C_DIS
LIN {X 111.74, Y 209.42, Z 0.00, A 0, B 0, C 0} C_DIS
LIN {X 111.53, Y 209.50, Z 0.00, A 0, B 0, C 0} C_DIS
LIN {X 111.32, Y 209.58, Z 0.00, A 0, B 0, C 0} C_DIS
LIN {X 111.11, Y 209.67, Z 0.00, A 0, B 0, C 0} C_DIS
LIN {X 110.90, Y 209.74, Z 0.00, A 0, B 0, C 0} C_DIS
LIN {X 110.68, Y 209.80, Z 0.00, A 0, B 0, C 0} C_DIS
LIN {X 110.47, Y 209.85, Z 0.00, A 0, B 0, C 0} C_DIS
LIN {X 110.25, Y 209.90, Z 0.00, A 0, B 0, C 0} C_DIS
LIN {X 110.04, Y 209.95, Z 0.00, A 0, B 0, C 0} C_DIS
LIN {X 109.83, Y 210.00, Z 0.00, A 0, B 0, C 0} C_DIS
LIN {X 109.61, Y 210.06, Z 0.00, A 0, B 0, C 0} C_DIS
LIN {X 109.40, Y 210.12, Z 0.00, A 0, B 0, C 0} C_DIS
LIN {X 109.19, Y 210.20, Z 0.00, A 0, B 0, C 0} C_DIS
LIN {X 108.97, Y 210.28, Z 0.00, A 0, B 0, C 0} C_DIS
LIN {X 108.77, Y 210.39, Z 0.00, A 0, B 0, C 0} C_DIS
LIN {X 108.57, Y 210.51, Z 0.00, A 0, B 0, C 0} C_DIS
LIN {X 108.37, Y 210.64, Z 0.00, A 0, B 0, C 0} C_DIS
LIN {X 108.17, Y 210.76, Z 0.00, A 0, B 0, C 0} C_DIS
LIN {X 107.96, Y 210.84, Z 0.00, A 0, B 0, C 0} C_DIS
LIN {X 107.74, Y 210.92, Z 0.00, A 0, B 0, C 0} C_DIS
LIN {X 107.53, Y 211.00, Z 0.00, A 0, B 0, C 0} C_DIS
LIN {X 107.33, Y 211.11, Z 0.00, A 0, B 0, C 0} C_DIS
LIN {X 107.14, Y 211.25, Z 0.00, A 0, B 0, C 0} C_DIS
LIN {X 106.94, Y 211.38, Z 0.00, A 0, B 0, C 0} C_DIS
LIN {X 106.72, Y 211.48, Z 0.00, A 0, B 0, C 0} C_DIS
LIN {X 106.49, Y 211.50, Z 0.00, A 0, B 0, C 0} C_DIS
LIN {X 106.31, Y 211.39, Z 0.00, A 0, B 0, C 0} C_DIS
LIN {X 106.20, Y 211.14, Z 0.00, A 0, B 0, C 0} C_DIS
LIN {X 106.14, Y 210.81, Z 0.00, A 0, B 0, C 0} C_DIS
LIN {X 106.12, Y 210.48, Z 0.00, A 0, B 0, C 0} C_DIS
LIN {X 106.12, Y 210.15, Z 0.00, A 0, B 0, C 0} C_DIS
LIN {X 106.12, Y 209.82, Z 0.00, A 0, B 0, C 0} C_DIS
LIN {X 106.12, Y 209.49, Z 0.00, A 0, B 0, C 0} C_DIS
LIN {X 106.12, Y 209.17, Z 0.00, A 0, B 0, C 0} C_DIS
LIN {X 106.12, Y 208.84, Z 0.00, A 0, B 0, C 0} C_DIS
LIN {X 106.12, Y 208.51, Z 0.00, A 0, B 0, C 0} C_DIS
LIN {X 106.12, Y 208.18, Z 0.00, A 0, B 0, C 0} C_DIS
LIN {X 106.12, Y 207.86, Z 0.00, A 0, B 0, C 0} C_DIS
LIN {X 106.12, Y 207.53, Z 0.00, A 0, B 0, C 0} C_DIS
LIN {X 106.12, Y 207.20, Z 0.00, A 0, B 0, C 0} C_DIS
LIN {X 106.13, Y 206.87, Z 0.00, A 0, B 0, C 0} C_DIS
LIN {X 106.13, Y 206.54, Z 0.00, A 0, B 0, C 0} C_DIS
LIN {X 106.13, Y 206.22, Z 0.00, A 0, B 0, C 0} C_DIS
LIN {X 106.12, Y 205.89, Z 0.00, A 0, B 0, C 0} C_DIS
LIN {X 106.10, Y 205.56, Z 0.00, A 0, B 0, C 0} C_DIS
LIN {X 106.08, Y 205.24, Z 0.00, A 0, B 0, C 0} C_DIS
LIN {X 106.04, Y 204.92, Z 0.00, A 0, B 0, C 0} C_DIS
LIN {X 106.00, Y 204.60, Z 0.00, A 0, B 0, C 0} C_DIS
LIN {X 105.94, Y 204.28, Z 0.00, A 0, B 0, C 0} C_DIS
LIN {X 105.88, Y 203.96, Z 0.00, A 0, B 0, C 0} C_DIS
LIN {X 105.82, Y 203.65, Z 0.00, A 0, B 0, C 0} C_DIS
LIN {X 105.77, Y 203.33, Z 0.00, A 0, B 0, C 0} C_DIS
LIN {X 105.73, Y 203.01, Z 0.00, A 0, B 0, C 0} C_DIS
LIN {X 105.70, Y 202.68, Z 0.00, A 0, B 0, C 0} C_DIS
LIN {X 105.68, Y 202.36, Z 0.00, A 0, B 0, C 0} C_DIS
LIN {X 105.68, Y 202.03, Z 0.00, A 0, B 0, C 0} C_DIS
LIN {X 105.69, Y 201.70, Z 0.00, A 0, B 0, C 0} C_DIS
LIN {X 105.69, Y 201.37, Z 0.00, A 0, B 0, C 0} C_DIS
LIN {X 105.70, Y 201.05, Z 0.00, A 0, B 0, C 0} C_DIS
LIN {X 105.69, Y 200.72, Z 0.00, A 0, B 0, C 0} C_DIS
LIN {X 105.68, Y 200.39, Z 0.00, A 0, B 0, C 0} C_DIS
LIN {X 105.65, Y 200.07, Z 0.00, A 0, B 0, C 0} C_DIS
LIN {X 105.62, Y 199.74, Z 0.00, A 0, B 0, C 0} C_DIS
LIN {X 105.57, Y 199.42, Z 0.00, A 0, B 0, C 0} C_DIS
LIN {X 105.52, Y 199.11, Z 0.00, A 0, B 0, C 0} C_DIS
LIN {X 105.45, Y 198.79, Z 0.00, A 0, B 0, C 0} C_DIS
LIN {X 105.39, Y 198.48, Z 0.00, A 0, B 0, C 0} C_DIS
LIN {X 105.34, Y 198.16, Z 0.00, A 0, B 0, C 0} C_DIS
LIN {X 105.31, Y 197.83, Z 0.00, A 0, B 0, C 0} C_DIS
LIN {X 105.28, Y 197.51, Z 0.00, A 0, B 0, C 0} C_DIS
LIN {X 105.25, Y 197.19, Z 0.00, A 0, B 0, C 0} C_DIS
LIN {X 105.22, Y 196.86, Z 0.00, A 0, B 0, C 0} C_DIS
LIN {X 105.18, Y 196.54, Z 0.00, A 0, B 0, C 0} C_DIS
LIN {X 105.14, Y 196.22, Z 0.00, A 0, B 0, C 0} C_DIS
LIN {X 105.09, Y 195.90, Z 0.00, A 0, B 0, C 0} C_DIS
LIN {X 105.04, Y 195.58, Z 0.00, A 0, B 0, C 0} C_DIS
LIN {X 104.99, Y 195.26, Z 0.00, A 0, B 0, C 0} C_DIS
LIN {X 104.93, Y 194.95, Z 0.00, A 0, B 0, C 0} C_DIS
LIN {X 104.88, Y 194.63, Z 0.00, A 0, B 0, C 0} C_DIS
LIN {X 104.82, Y 194.31, Z 0.00, A 0, B 0, C 0} C_DIS
LIN {X 104.77, Y 193.99, Z 0.00, A 0, B 0, C 0} C_DIS
LIN {X 104.72, Y 193.68, Z 0.00, A 0, B 0, C 0} C_DIS
LIN {X 104.67, Y 193.36, Z 0.00, A 0, B 0, C 0} C_DIS
LIN {X 104.61, Y 193.04, Z 0.00, A 0, B 0, C 0} C_DIS
LIN {X 104.55, Y 192.72, Z 0.00, A 0, B 0, C 0} C_DIS
LIN {X 104.49, Y 192.41, Z 0.00, A 0, B 0, C 0} C_DIS
LIN {X 104.42, Y 192.10, Z 0.00, A 0, B 0, C 0} C_DIS
LIN {X 104.35, Y 191.80, Z 0.00, A 0, B 0, C 0} C_DIS
LIN {X 104.26, Y 191.49, Z 0.00, A 0, B 0, C 0} C_DIS
LIN {X 104.19, Y 191.19, Z 0.00, A 0, B 0, C 0} C_DIS
LIN {X 104.13, Y 190.87, Z 0.00, A 0, B 0, C 0} C_DIS
LIN {X 104.09, Y 190.55, Z 0.00, A 0, B 0, C 0} C_DIS
LIN {X 104.02, Y 190.24, Z 0.00, A 0, B 0, C 0} C_DIS
LIN {X 103.93, Y 189.94, Z 0.00, A 0, B 0, C 0} C_DIS
LIN {X 103.84, Y 189.64, Z 0.00, A 0, B 0, C 0} C_DIS
LIN {X 103.77, Y 189.33, Z 0.00, A 0, B 0, C 0} C_DIS
LIN {X 103.72, Y 189.01, Z 0.00, A 0, B 0, C 0} C_DIS
LIN {X 103.67, Y 188.69, Z 0.00, A 0, B 0, C 0} C_DIS
LIN {X 103.61, Y 188.38, Z 0.00, A 0, B 0, C 0} C_DIS
LIN {X 103.53, Y 188.08, Z 0.00, A 0, B 0, C 0} C_DIS
LIN {X 103.44, Y 187.78, Z 0.00, A 0, B 0, C 0} C_DIS
LIN {X 103.36, Y 187.47, Z 0.00, A 0, B 0, C 0} C_DIS
LIN {X 103.30, Y 187.16, Z 0.00, A 0, B 0, C 0} C_DIS
LIN {X 103.24, Y 186.84, Z 0.00, A 0, B 0, C 0} C_DIS
LIN {X 103.15, Y 186.55, Z 0.00, A 0, B 0, C 0} C_DIS
LIN {X 103.03, Y 186.27, Z 0.00, A 0, B 0, C 0} C_DIS
LIN {X 102.92, Y 185.99, Z 0.00, A 0, B 0, C 0} C_DIS
LIN {X 102.85, Y 185.68, Z 0.00, A 0, B 0, C 0} C_DIS
LIN {X 102.80, Y 185.36, Z 0.00, A 0, B 0, C 0} C_DIS
LIN {X 102.73, Y 185.05, Z 0.00, A 0, B 0, C 0} C_DIS
LIN {X 102.64, Y 184.75, Z 0.00, A 0, B 0, C 0} C_DIS
LIN {X 102.55, Y 184.45, Z 0.00, A 0, B 0, C 0} C_DIS
LIN {X 102.48, Y 184.14, Z 0.00, A 0, B 0, C 0} C_DIS
LIN {X 102.43, Y 183.82, Z 0.00, A 0, B 0, C 0} C_DIS
LIN {X 102.36, Y 183.52, Z 0.00, A 0, B 0, C 0} C_DIS
LIN {X 102.26, Y 183.23, Z 0.00, A 0, B 0, C 0} C_DIS
LIN {X 102.14, Y 182.95, Z 0.00, A 0, B 0, C 0} C_DIS
LIN {X 102.04, Y 182.66, Z 0.00, A 0, B 0, C 0} C_DIS
LIN {X 101.96, Y 182.35, Z 0.00, A 0, B 0, C 0} C_DIS
LIN {X 101.87, Y 182.06, Z 0.00, A 0, B 0, C 0} C_DIS
LIN {X 101.76, Y 181.77, Z 0.00, A 0, B 0, C 0} C_DIS
LIN {X 101.66, Y 181.49, Z 0.00, A 0, B 0, C 0} C_DIS
LIN {X 101.57, Y 181.19, Z 0.00, A 0, B 0, C 0} C_DIS
LIN {X 101.48, Y 180.89, Z 0.00, A 0, B 0, C 0} C_DIS
LIN {X 101.38, Y 180.60, Z 0.00, A 0, B 0, C 0} C_DIS
LIN {X 101.27, Y 180.32, Z 0.00, A 0, B 0, C 0} C_DIS
LIN {X 101.18, Y 180.03, Z 0.00, A 0, B 0, C 0} C_DIS
LIN {X 101.09, Y 179.73, Z 0.00, A 0, B 0, C 0} C_DIS
LIN {X 100.99, Y 179.43, Z 0.00, A 0, B 0, C 0} C_DIS
LIN {X 100.89, Y 179.15, Z 0.00, A 0, B 0, C 0} C_DIS
LIN {X 100.78, Y 178.87, Z 0.00, A 0, B 0, C 0} C_DIS
LIN {X 100.66, Y 178.59, Z 0.00, A 0, B 0, C 0} C_DIS
LIN {X 100.53, Y 178.33, Z 0.00, A 0, B 0, C 0} C_DIS
LIN {X 100.40, Y 178.06, Z 0.00, A 0, B 0, C 0} C_DIS
LIN {X 100.28, Y 177.79, Z 0.00, A 0, B 0, C 0} C_DIS
LIN {X 100.16, Y 177.52, Z 0.00, A 0, B 0, C 0} C_DIS
LIN {X 100.05, Y 177.24, Z 0.00, A 0, B 0, C 0} C_DIS
LIN {X 99.94, Y 176.95, Z 0.00, A 0, B 0, C 0} C_DIS
LIN {X 99.85, Y 176.66, Z 0.00, A 0, B 0, C 0} C_DIS
LIN {X 99.75, Y 176.37, Z 0.00, A 0, B 0, C 0} C_DIS
LIN {X 99.65, Y 176.07, Z 0.00, A 0, B 0, C 0} C_DIS
LIN {X 99.55, Y 175.79, Z 0.00, A 0, B 0, C 0} C_DIS
LIN {X 99.44, Y 175.50, Z 0.00, A 0, B 0, C 0} C_DIS
LIN {X 99.32, Y 175.23, Z 0.00, A 0, B 0, C 0} C_DIS
LIN {X 99.18, Y 174.97, Z 0.00, A 0, B 0, C 0} C_DIS
LIN {X 99.04, Y 174.73, Z 0.00, A 0, B 0, C 0} C_DIS
LIN {X 98.89, Y 174.49, Z 0.00, A 0, B 0, C 0} C_DIS
LIN {X 98.74, Y 174.26, Z 0.00, A 0, B 0, C 0} C_DIS
LIN {X 98.61, Y 174.00, Z 0.00, A 0, B 0, C 0} C_DIS
LIN {X 98.49, Y 173.72, Z 0.00, A 0, B 0, C 0} C_DIS
LIN {X 98.37, Y 173.45, Z 0.00, A 0, B 0, C 0} C_DIS
LIN {X 98.25, Y 173.17, Z 0.00, A 0, B 0, C 0} C_DIS
LIN {X 98.13, Y 172.91, Z 0.00, A 0, B 0, C 0} C_DIS
LIN {X 98.00, Y 172.64, Z 0.00, A 0, B 0, C 0} C_DIS
LIN {X 97.88, Y 172.37, Z 0.00, A 0, B 0, C 0} C_DIS
LIN {X 97.76, Y 172.09, Z 0.00, A 0, B 0, C 0} C_DIS
LIN {X 97.65, Y 171.81, Z 0.00, A 0, B 0, C 0} C_DIS
LIN {X 97.53, Y 171.54, Z 0.00, A 0, B 0, C 0} C_DIS
LIN {X 97.41, Y 171.26, Z 0.00, A 0, B 0, C 0} C_DIS
LIN {X 97.29, Y 170.98, Z 0.00, A 0, B 0, C 0} C_DIS
LIN {X 97.17, Y 170.72, Z 0.00, A 0, B 0, C 0} C_DIS
LIN {X 97.04, Y 170.46, Z 0.00, A 0, B 0, C 0} C_DIS
LIN {X 96.90, Y 170.20, Z 0.00, A 0, B 0, C 0} C_DIS
LIN {X 96.76, Y 169.96, Z 0.00, A 0, B 0, C 0} C_DIS
LIN {X 96.60, Y 169.73, Z 0.00, A 0, B 0, C 0} C_DIS
LIN {X 96.45, Y 169.50, Z 0.00, A 0, B 0, C 0} C_DIS
LIN {X 96.29, Y 169.27, Z 0.00, A 0, B 0, C 0} C_DIS
LIN {X 96.14, Y 169.04, Z 0.00, A 0, B 0, C 0} C_DIS
LIN {X 95.99, Y 168.80, Z 0.00, A 0, B 0, C 0} C_DIS
LIN {X 95.84, Y 168.57, Z 0.00, A 0, B 0, C 0} C_DIS
LIN {X 95.68, Y 168.33, Z 0.00, A 0, B 0, C 0} C_DIS
LIN {X 95.52, Y 168.11, Z 0.00, A 0, B 0, C 0} C_DIS
LIN {X 95.36, Y 167.90, Z 0.00, A 0, B 0, C 0} C_DIS
LIN {X 95.18, Y 167.71, Z 0.00, A 0, B 0, C 0} C_DIS
LIN {X 95.00, Y 167.53, Z 0.00, A 0, B 0, C 0} C_DIS
LIN {X 94.82, Y 167.35, Z 0.00, A 0, B 0, C 0} C_DIS
LIN {X 94.63, Y 167.19, Z 0.00, A 0, B 0, C 0} C_DIS
LIN {X 94.43, Y 167.08, Z 0.00, A 0, B 0, C 0} C_DIS
LIN {X 94.21, Y 167.04, Z 0.00, A 0, B 0, C 0} C_DIS
LIN {X 93.99, Y 167.05, Z 0.00, A 0, B 0, C 0} C_DIS
LIN {X 93.78, Y 167.10, Z 0.00, A 0, B 0, C 0} C_DIS
LIN {X 93.58, Y 167.21, Z 0.00, A 0, B 0, C 0} C_DIS
LIN {X 93.39, Y 167.37, Z 0.00, A 0, B 0, C 0} C_DIS
LIN {X 93.20, Y 167.55, Z 0.00, A 0, B 0, C 0} C_DIS
LIN {X 93.03, Y 167.74, Z 0.00, A 0, B 0, C 0} C_DIS
LIN {X 92.86, Y 167.94, Z 0.00, A 0, B 0, C 0} C_DIS
LIN {X 92.69, Y 168.15, Z 0.00, A 0, B 0, C 0} C_DIS
LIN {X 92.53, Y 168.37, Z 0.00, A 0, B 0, C 0} C_DIS
LIN {X 92.37, Y 168.60, Z 0.00, A 0, B 0, C 0} C_DIS
LIN {X 92.22, Y 168.83, Z 0.00, A 0, B 0, C 0} C_DIS
LIN {X 92.07, Y 169.07, Z 0.00, A 0, B 0, C 0} C_DIS
LIN {X 91.92, Y 169.30, Z 0.00, A 0, B 0, C 0} C_DIS
LIN {X 91.77, Y 169.54, Z 0.00, A 0, B 0, C 0} C_DIS
LIN {X 91.61, Y 169.77, Z 0.00, A 0, B 0, C 0} C_DIS
LIN {X 91.46, Y 170.00, Z 0.00, A 0, B 0, C 0} C_DIS
LIN {X 91.31, Y 170.23, Z 0.00, A 0, B 0, C 0} C_DIS
LIN {X 91.15, Y 170.46, Z 0.00, A 0, B 0, C 0} C_DIS
LIN {X 91.00, Y 170.69, Z 0.00, A 0, B 0, C 0} C_DIS
LIN {X 90.84, Y 170.92, Z 0.00, A 0, B 0, C 0} C_DIS
LIN {X 90.68, Y 171.15, Z 0.00, A 0, B 0, C 0} C_DIS
LIN {X 90.53, Y 171.38, Z 0.00, A 0, B 0, C 0} C_DIS
LIN {X 90.37, Y 171.61, Z 0.00, A 0, B 0, C 0} C_DIS
LIN {X 90.22, Y 171.85, Z 0.00, A 0, B 0, C 0} C_DIS
LIN {X 90.08, Y 172.09, Z 0.00, A 0, B 0, C 0} C_DIS
LIN {X 89.94, Y 172.34, Z 0.00, A 0, B 0, C 0} C_DIS
LIN {X 89.80, Y 172.59, Z 0.00, A 0, B 0, C 0} C_DIS
LIN {X 89.68, Y 172.87, Z 0.00, A 0, B 0, C 0} C_DIS
LIN {X 89.56, Y 173.14, Z 0.00, A 0, B 0, C 0} C_DIS
LIN {X 89.44, Y 173.42, Z 0.00, A 0, B 0, C 0} C_DIS
LIN {X 89.35, Y 173.71, Z 0.00, A 0, B 0, C 0} C_DIS
LIN {X 89.29, Y 174.02, Z 0.00, A 0, B 0, C 0} C_DIS
LIN {X 89.26, Y 174.34, Z 0.00, A 0, B 0, C 0} C_DIS
LIN {X 89.25, Y 174.68, Z 0.00, A 0, B 0, C 0} C_DIS
LIN {X 89.27, Y 175.01, Z 0.00, A 0, B 0, C 0} C_DIS
LIN {X 89.32, Y 175.33, Z 0.00, A 0, B 0, C 0} C_DIS
LIN {X 89.41, Y 175.62, Z 0.00, A 0, B 0, C 0} C_DIS
LIN {X 89.52, Y 175.90, Z 0.00, A 0, B 0, C 0} C_DIS
LIN {X 89.63, Y 176.19, Z 0.00, A 0, B 0, C 0} C_DIS
LIN {X 89.72, Y 176.49, Z 0.00, A 0, B 0, C 0} C_DIS
LIN {X 89.80, Y 176.79, Z 0.00, A 0, B 0, C 0} C_DIS
LIN {X 89.90, Y 177.08, Z 0.00, A 0, B 0, C 0} C_DIS
LIN {X 90.01, Y 177.36, Z 0.00, A 0, B 0, C 0} C_DIS
LIN {X 90.13, Y 177.63, Z 0.00, A 0, B 0, C 0} C_DIS
LIN {X 90.26, Y 177.90, Z 0.00, A 0, B 0, C 0} C_DIS
LIN {X 90.39, Y 178.16, Z 0.00, A 0, B 0, C 0} C_DIS
LIN {X 90.53, Y 178.41, Z 0.00, A 0, B 0, C 0} C_DIS
LIN {X 90.68, Y 178.64, Z 0.00, A 0, B 0, C 0} C_DIS
LIN {X 90.83, Y 178.87, Z 0.00, A 0, B 0, C 0} C_DIS
LIN {X 90.99, Y 179.10, Z 0.00, A 0, B 0, C 0} C_DIS
LIN {X 91.14, Y 179.34, Z 0.00, A 0, B 0, C 0} C_DIS
LIN {X 91.28, Y 179.58, Z 0.00, A 0, B 0, C 0} C_DIS
LIN {X 91.42, Y 179.84, Z 0.00, A 0, B 0, C 0} C_DIS
LIN {X 91.54, Y 180.11, Z 0.00, A 0, B 0, C 0} C_DIS
LIN {X 91.66, Y 180.38, Z 0.00, A 0, B 0, C 0} C_DIS
LIN {X 91.78, Y 180.66, Z 0.00, A 0, B 0, C 0} C_DIS
LIN {X 91.89, Y 180.94, Z 0.00, A 0, B 0, C 0} C_DIS
LIN {X 92.01, Y 181.22, Z 0.00, A 0, B 0, C 0} C_DIS
LIN {X 92.13, Y 181.49, Z 0.00, A 0, B 0, C 0} C_DIS
LIN {X 92.25, Y 181.76, Z 0.00, A 0, B 0, C 0} C_DIS
LIN {X 92.38, Y 182.03, Z 0.00, A 0, B 0, C 0} C_DIS
LIN {X 92.50, Y 182.30, Z 0.00, A 0, B 0, C 0} C_DIS
LIN {X 92.62, Y 182.57, Z 0.00, A 0, B 0, C 0} C_DIS
LIN {X 92.74, Y 182.84, Z 0.00, A 0, B 0, C 0} C_DIS
LIN {X 92.86, Y 183.12, Z 0.00, A 0, B 0, C 0} C_DIS
LIN {X 92.98, Y 183.39, Z 0.00, A 0, B 0, C 0} C_DIS
LIN {X 93.10, Y 183.67, Z 0.00, A 0, B 0, C 0} C_DIS
LIN {X 93.22, Y 183.94, Z 0.00, A 0, B 0, C 0} C_DIS
LIN {X 93.35, Y 184.20, Z 0.00, A 0, B 0, C 0} C_DIS
LIN {X 93.46, Y 184.48, Z 0.00, A 0, B 0, C 0} C_DIS
LIN {X 93.56, Y 184.77, Z 0.00, A 0, B 0, C 0} C_DIS
LIN {X 93.65, Y 185.07, Z 0.00, A 0, B 0, C 0} C_DIS
LIN {X 93.74, Y 185.37, Z 0.00, A 0, B 0, C 0} C_DIS
LIN {X 93.84, Y 185.66, Z 0.00, A 0, B 0, C 0} C_DIS
LIN {X 93.95, Y 185.94, Z 0.00, A 0, B 0, C 0} C_DIS
LIN {X 94.04, Y 186.24, Z 0.00, A 0, B 0, C 0} C_DIS
LIN {X 94.13, Y 186.54, Z 0.00, A 0, B 0, C 0} C_DIS
LIN {X 94.23, Y 186.83, Z 0.00, A 0, B 0, C 0} C_DIS
LIN {X 94.33, Y 187.11, Z 0.00, A 0, B 0, C 0} C_DIS
LIN {X 94.43, Y 187.40, Z 0.00, A 0, B 0, C 0} C_DIS
LIN {X 94.52, Y 187.70, Z 0.00, A 0, B 0, C 0} C_DIS
LIN {X 94.61, Y 188.00, Z 0.00, A 0, B 0, C 0} C_DIS
LIN {X 94.71, Y 188.29, Z 0.00, A 0, B 0, C 0} C_DIS
LIN {X 94.82, Y 188.57, Z 0.00, A 0, B 0, C 0} C_DIS
LIN {X 94.92, Y 188.86, Z 0.00, A 0, B 0, C 0} C_DIS
LIN {X 95.00, Y 189.16, Z 0.00, A 0, B 0, C 0} C_DIS
LIN {X 95.09, Y 189.46, Z 0.00, A 0, B 0, C 0} C_DIS
LIN {X 95.20, Y 189.74, Z 0.00, A 0, B 0, C 0} C_DIS
LIN {X 95.31, Y 190.03, Z 0.00, A 0, B 0, C 0} C_DIS
LIN {X 95.39, Y 190.32, Z 0.00, A 0, B 0, C 0} C_DIS
LIN {X 95.45, Y 190.64, Z 0.00, A 0, B 0, C 0} C_DIS
LIN {X 95.51, Y 190.96, Z 0.00, A 0, B 0, C 0} C_DIS
LIN {X 95.59, Y 191.26, Z 0.00, A 0, B 0, C 0} C_DIS
LIN {X 95.68, Y 191.56, Z 0.00, A 0, B 0, C 0} C_DIS
LIN {X 95.76, Y 191.87, Z 0.00, A 0, B 0, C 0} C_DIS
LIN {X 95.81, Y 192.18, Z 0.00, A 0, B 0, C 0} C_DIS
LIN {X 95.86, Y 192.50, Z 0.00, A 0, B 0, C 0} C_DIS
LIN {X 95.92, Y 192.82, Z 0.00, A 0, B 0, C 0} C_DIS
LIN {X 96.00, Y 193.12, Z 0.00, A 0, B 0, C 0} C_DIS
LIN {X 96.09, Y 193.42, Z 0.00, A 0, B 0, C 0} C_DIS
LIN {X 96.17, Y 193.72, Z 0.00, A 0, B 0, C 0} C_DIS
LIN {X 96.23, Y 194.04, Z 0.00, A 0, B 0, C 0} C_DIS
LIN {X 96.28, Y 194.36, Z 0.00, A 0, B 0, C 0} C_DIS
LIN {X 96.33, Y 194.68, Z 0.00, A 0, B 0, C 0} C_DIS
LIN {X 96.40, Y 194.99, Z 0.00, A 0, B 0, C 0} C_DIS
LIN {X 96.49, Y 195.29, Z 0.00, A 0, B 0, C 0} C_DIS
LIN {X 96.57, Y 195.59, Z 0.00, A 0, B 0, C 0} C_DIS
LIN {X 96.65, Y 195.89, Z 0.00, A 0, B 0, C 0} C_DIS
LIN {X 96.71, Y 196.21, Z 0.00, A 0, B 0, C 0} C_DIS
LIN {X 96.76, Y 196.53, Z 0.00, A 0, B 0, C 0} C_DIS
LIN {X 96.80, Y 196.85, Z 0.00, A 0, B 0, C 0} C_DIS
LIN {X 96.84, Y 197.17, Z 0.00, A 0, B 0, C 0} C_DIS
LIN {X 96.87, Y 197.50, Z 0.00, A 0, B 0, C 0} C_DIS
LIN {X 96.90, Y 197.82, Z 0.00, A 0, B 0, C 0} C_DIS
LIN {X 96.94, Y 198.14, Z 0.00, A 0, B 0, C 0} C_DIS
LIN {X 96.97, Y 198.47, Z 0.00, A 0, B 0, C 0} C_DIS
LIN {X 97.01, Y 198.79, Z 0.00, A 0, B 0, C 0} C_DIS
LIN {X 97.05, Y 199.11, Z 0.00, A 0, B 0, C 0} C_DIS
LIN {X 97.11, Y 199.43, Z 0.00, A 0, B 0, C 0} C_DIS
LIN {X 97.17, Y 199.74, Z 0.00, A 0, B 0, C 0} C_DIS
LIN {X 97.23, Y 200.06, Z 0.00, A 0, B 0, C 0} C_DIS
LIN {X 97.28, Y 200.38, Z 0.00, A 0, B 0, C 0} C_DIS
LIN {X 97.32, Y 200.70, Z 0.00, A 0, B 0, C 0} C_DIS
LIN {X 97.33, Y 201.02, Z 0.00, A 0, B 0, C 0} C_DIS
LIN {X 97.33, Y 201.35, Z 0.00, A 0, B 0, C 0} C_DIS
LIN {X 97.34, Y 201.68, Z 0.00, A 0, B 0, C 0} C_DIS
LIN {X 97.35, Y 202.01, Z 0.00, A 0, B 0, C 0} C_DIS
LIN {X 97.38, Y 202.33, Z 0.00, A 0, B 0, C 0} C_DIS
LIN {X 97.43, Y 202.65, Z 0.00, A 0, B 0, C 0} C_DIS
LIN {X 97.48, Y 202.97, Z 0.00, A 0, B 0, C 0} C_DIS
LIN {X 97.54, Y 203.29, Z 0.00, A 0, B 0, C 0} C_DIS
LIN {X 97.60, Y 203.60, Z 0.00, A 0, B 0, C 0} C_DIS
LIN {X 97.66, Y 203.92, Z 0.00, A 0, B 0, C 0} C_DIS
LIN {X 97.70, Y 204.24, Z 0.00, A 0, B 0, C 0} C_DIS
LIN {X 97.73, Y 204.56, Z 0.00, A 0, B 0, C 0} C_DIS
LIN {X 97.76, Y 204.89, Z 0.00, A 0, B 0, C 0} C_DIS
LIN {X 97.77, Y 205.21, Z 0.00, A 0, B 0, C 0} C_DIS
LIN {X 97.78, Y 205.54, Z 0.00, A 0, B 0, C 0} C_DIS
LIN {X 97.78, Y 205.87, Z 0.00, A 0, B 0, C 0} C_DIS
LIN {X 97.78, Y 206.19, Z 0.00, A 0, B 0, C 0} C_DIS
LIN {X 97.78, Y 206.52, Z 0.00, A 0, B 0, C 0} C_DIS
LIN {X 97.77, Y 206.85, Z 0.00, A 0, B 0, C 0} C_DIS
LIN {X 97.77, Y 207.18, Z 0.00, A 0, B 0, C 0} C_DIS
LIN {X 97.77, Y 207.51, Z 0.00, A 0, B 0, C 0} C_DIS
LIN {X 97.77, Y 207.84, Z 0.00, A 0, B 0, C 0} C_DIS
LIN {X 97.77, Y 208.16, Z 0.00, A 0, B 0, C 0} C_DIS
LIN {X 97.77, Y 208.49, Z 0.00, A 0, B 0, C 0} C_DIS
LIN {X 97.77, Y 208.82, Z 0.00, A 0, B 0, C 0} C_DIS
LIN {X 97.77, Y 209.15, Z 0.00, A 0, B 0, C 0} C_DIS
LIN {X 97.77, Y 209.47, Z 0.00, A 0, B 0, C 0} C_DIS
LIN {X 97.77, Y 209.80, Z 0.00, A 0, B 0, C 0} C_DIS
LIN {X 97.77, Y 210.13, Z 0.00, A 0, B 0, C 0} C_DIS
LIN {X 97.77, Y 210.46, Z 0.00, A 0, B 0, C 0} C_DIS
LIN {X 97.77, Y 210.78, Z 0.00, A 0, B 0, C 0} C_DIS
LIN {X 97.77, Y 211.11, Z 0.00, A 0, B 0, C 0} C_DIS
LIN {X 97.77, Y 211.44, Z 0.00, A 0, B 0, C 0} C_DIS
LIN {X 97.77, Y 211.77, Z 0.00, A 0, B 0, C 0} C_DIS
LIN {X 97.77, Y 212.09, Z 0.00, A 0, B 0, C 0} C_DIS
LIN {X 97.77, Y 212.42, Z 0.00, A 0, B 0, C 0} C_DIS
LIN {X 97.77, Y 212.75, Z 0.00, A 0, B 0, C 0} C_DIS
LIN {X 97.77, Y 213.08, Z 0.00, A 0, B 0, C 0} C_DIS
LIN {X 97.77, Y 213.41, Z 0.00, A 0, B 0, C 0} C_DIS
LIN {X 97.76, Y 213.73, Z 0.00, A 0, B 0, C 0} C_DIS
LIN {X 97.74, Y 214.06, Z 0.00, A 0, B 0, C 0} C_DIS
LIN {X 97.71, Y 214.38, Z 0.00, A 0, B 0, C 0} C_DIS
LIN {X 97.66, Y 214.70, Z 0.00, A 0, B 0, C 0} C_DIS
LIN {X 97.60, Y 215.02, Z 0.00, A 0, B 0, C 0} C_DIS
LIN {X 97.54, Y 215.33, Z 0.00, A 0, B 0, C 0} C_DIS
LIN {X 97.48, Y 215.65, Z 0.00, A 0, B 0, C 0} C_DIS
LIN {X 97.43, Y 215.97, Z 0.00, A 0, B 0, C 0} C_DIS
LIN {X 97.39, Y 216.29, Z 0.00, A 0, B 0, C 0} C_DIS
LIN {X 97.36, Y 216.61, Z 0.00, A 0, B 0, C 0} C_DIS
LIN {X 97.33, Y 216.94, Z 0.00, A 0, B 0, C 0} C_DIS
LIN {X 97.31, Y 217.26, Z 0.00, A 0, B 0, C 0} C_DIS
LIN {X 97.27, Y 217.59, Z 0.00, A 0, B 0, C 0} C_DIS
LIN {X 97.23, Y 217.91, Z 0.00, A 0, B 0, C 0} C_DIS
LIN {X 97.18, Y 218.22, Z 0.00, A 0, B 0, C 0} C_DIS
LIN {X 97.12, Y 218.54, Z 0.00, A 0, B 0, C 0} C_DIS
LIN {X 97.06, Y 218.86, Z 0.00, A 0, B 0, C 0} C_DIS
LIN {X 97.00, Y 219.17, Z 0.00, A 0, B 0, C 0} C_DIS
LIN {X 96.96, Y 219.49, Z 0.00, A 0, B 0, C 0} C_DIS
LIN {X 96.93, Y 219.82, Z 0.00, A 0, B 0, C 0} C_DIS
LIN {X 96.91, Y 220.14, Z 0.00, A 0, B 0, C 0} C_DIS
LIN {X 96.90, Y 220.47, Z 0.00, A 0, B 0, C 0} C_DIS
LIN {X 96.89, Y 220.80, Z 0.00, A 0, B 0, C 0} C_DIS
LIN {X 96.88, Y 221.12, Z 0.00, A 0, B 0, C 0} C_DIS
LIN {X 96.85, Y 221.45, Z 0.00, A 0, B 0, C 0} C_DIS
LIN {X 96.81, Y 221.77, Z 0.00, A 0, B 0, C 0} C_DIS
LIN {X 96.76, Y 222.09, Z 0.00, A 0, B 0, C 0} C_DIS
LIN {X 96.70, Y 222.40, Z 0.00, A 0, B 0, C 0} C_DIS
LIN {X 96.63, Y 222.72, Z 0.00, A 0, B 0, C 0} C_DIS
LIN {X 96.57, Y 223.03, Z 0.00, A 0, B 0, C 0} C_DIS
LIN {X 96.49, Y 223.33, Z 0.00, A 0, B 0, C 0} C_DIS
LIN {X 96.42, Y 223.64, Z 0.00, A 0, B 0, C 0} C_DIS
LIN {X 96.34, Y 223.95, Z 0.00, A 0, B 0, C 0} C_DIS
LIN {X 96.27, Y 224.26, Z 0.00, A 0, B 0, C 0} C_DIS
LIN {X 96.22, Y 224.57, Z 0.00, A 0, B 0, C 0} C_DIS
LIN {X 96.16, Y 224.89, Z 0.00, A 0, B 0, C 0} C_DIS
LIN {X 96.10, Y 225.20, Z 0.00, A 0, B 0, C 0} C_DIS
LIN {X 96.01, Y 225.50, Z 0.00, A 0, B 0, C 0} C_DIS
LIN {X 95.92, Y 225.80, Z 0.00, A 0, B 0, C 0} C_DIS
LIN {X 95.85, Y 226.11, Z 0.00, A 0, B 0, C 0} C_DIS
LIN {X 95.81, Y 226.43, Z 0.00, A 0, B 0, C 0} C_DIS
LIN {X 95.76, Y 226.75, Z 0.00, A 0, B 0, C 0} C_DIS
LIN {X 95.69, Y 227.06, Z 0.00, A 0, B 0, C 0} C_DIS
LIN {X 95.60, Y 227.36, Z 0.00, A 0, B 0, C 0} C_DIS
LIN {X 95.51, Y 227.66, Z 0.00, A 0, B 0, C 0} C_DIS
LIN {X 95.45, Y 227.97, Z 0.00, A 0, B 0, C 0} C_DIS
LIN {X 95.39, Y 228.29, Z 0.00, A 0, B 0, C 0} C_DIS
LIN {X 95.31, Y 228.59, Z 0.00, A 0, B 0, C 0} C_DIS
LIN {X 95.21, Y 228.88, Z 0.00, A 0, B 0, C 0} C_DIS
LIN {X 95.10, Y 229.17, Z 0.00, A 0, B 0, C 0} C_DIS
LIN {X 95.00, Y 229.45, Z 0.00, A 0, B 0, C 0} C_DIS
LIN {X 94.91, Y 229.75, Z 0.00, A 0, B 0, C 0} C_DIS
LIN {X 94.83, Y 230.05, Z 0.00, A 0, B 0, C 0} C_DIS
LIN {X 94.72, Y 230.33, Z 0.00, A 0, B 0, C 0} C_DIS
LIN {X 94.61, Y 230.62, Z 0.00, A 0, B 0, C 0} C_DIS
LIN {X 94.52, Y 230.92, Z 0.00, A 0, B 0, C 0} C_DIS
LIN {X 94.44, Y 231.22, Z 0.00, A 0, B 0, C 0} C_DIS
LIN {X 94.34, Y 231.51, Z 0.00, A 0, B 0, C 0} C_DIS
LIN {X 94.23, Y 231.79, Z 0.00, A 0, B 0, C 0} C_DIS
LIN {X 94.13, Y 232.08, Z 0.00, A 0, B 0, C 0} C_DIS
LIN {X 94.04, Y 232.38, Z 0.00, A 0, B 0, C 0} C_DIS
LIN {X 93.95, Y 232.68, Z 0.00, A 0, B 0, C 0} C_DIS
LIN {X 93.85, Y 232.97, Z 0.00, A 0, B 0, C 0} C_DIS
LIN {X 93.74, Y 233.25, Z 0.00, A 0, B 0, C 0} C_DIS
LIN {X 93.65, Y 233.54, Z 0.00, A 0, B 0, C 0} C_DIS
LIN {X 93.56, Y 233.85, Z 0.00, A 0, B 0, C 0} C_DIS
LIN {X 93.46, Y 234.14, Z 0.00, A 0, B 0, C 0} C_DIS
LIN {X 93.35, Y 234.42, Z 0.00, A 0, B 0, C 0} C_DIS
LIN {X 93.26, Y 234.71, Z 0.00, A 0, B 0, C 0} C_DIS
LIN {X 93.17, Y 235.01, Z 0.00, A 0, B 0, C 0} C_DIS
LIN {X 93.08, Y 235.31, Z 0.00, A 0, B 0, C 0} C_DIS
LIN {X 92.97, Y 235.59, Z 0.00, A 0, B 0, C 0} C_DIS
LIN {X 92.87, Y 235.88, Z 0.00, A 0, B 0, C 0} C_DIS
LIN {X 92.78, Y 236.18, Z 0.00, A 0, B 0, C 0} C_DIS
LIN {X 92.69, Y 236.48, Z 0.00, A 0, B 0, C 0} C_DIS
LIN {X 92.59, Y 236.76, Z 0.00, A 0, B 0, C 0} C_DIS
LIN {X 92.48, Y 237.04, Z 0.00, A 0, B 0, C 0} C_DIS
LIN {X 92.39, Y 237.34, Z 0.00, A 0, B 0, C 0} C_DIS
LIN {X 92.30, Y 237.64, Z 0.00, A 0, B 0, C 0} C_DIS
LIN {X 92.21, Y 237.94, Z 0.00, A 0, B 0, C 0} C_DIS
LIN {X 92.10, Y 238.22, Z 0.00, A 0, B 0, C 0} C_DIS
LIN {X 91.99, Y 238.50, Z 0.00, A 0, B 0, C 0} C_DIS
LIN {X 91.91, Y 238.80, Z 0.00, A 0, B 0, C 0} C_DIS
LIN {X 91.82, Y 239.10, Z 0.00, A 0, B 0, C 0} C_DIS
LIN {X 91.72, Y 239.39, Z 0.00, A 0, B 0, C 0} C_DIS
LIN {X 91.61, Y 239.67, Z 0.00, A 0, B 0, C 0} C_DIS
LIN {X 91.51, Y 239.97, Z 0.00, A 0, B 0, C 0} C_DIS
LIN {X 91.43, Y 240.27, Z 0.00, A 0, B 0, C 0} C_DIS
LIN {X 91.34, Y 240.57, Z 0.00, A 0, B 0, C 0} C_DIS
LIN {X 91.22, Y 240.84, Z 0.00, A 0, B 0, C 0} C_DIS
LIN {X 91.12, Y 241.13, Z 0.00, A 0, B 0, C 0} C_DIS
LIN {X 91.04, Y 241.43, Z 0.00, A 0, B 0, C 0} C_DIS
LIN {X 91.00, Y 241.75, Z 0.00, A 0, B 0, C 0} C_DIS
LIN {X 90.99, Y 242.08, Z 0.00, A 0, B 0, C 0} C_DIS
LIN {X 91.01, Y 242.42, Z 0.00, A 0, B 0, C 0} C_DIS
LIN {X 91.05, Y 242.74, Z 0.00, A 0, B 0, C 0} C_DIS
LIN {X 91.11, Y 243.04, Z 0.00, A 0, B 0, C 0} C_DIS
LIN {X 91.23, Y 243.31, Z 0.00, A 0, B 0, C 0} C_DIS
LIN {X 91.38, Y 243.55, Z 0.00, A 0, B 0, C 0} C_DIS
LIN {X 91.54, Y 243.78, Z 0.00, A 0, B 0, C 0} C_DIS
LIN {X 91.70, Y 244.01, Z 0.00, A 0, B 0, C 0} C_DIS
LIN {X 91.86, Y 244.23, Z 0.00, A 0, B 0, C 0} C_DIS
LIN {X 92.04, Y 244.38, Z 0.00, A 0, B 0, C 0} C_DIS
LIN {X 92.25, Y 244.47, Z 0.00, A 0, B 0, C 0} C_DIS
LIN {X 92.47, Y 244.55, Z 0.00, A 0, B 0, C 0} C_DIS
LIN {X 92.67, Y 244.66, Z 0.00, A 0, B 0, C 0} C_DIS
LIN {X 92.87, Y 244.80, Z 0.00, A 0, B 0, C 0} C_DIS
LIN {X 93.07, Y 244.92, Z 0.00, A 0, B 0, C 0} C_DIS
LIN {X 93.28, Y 245.02, Z 0.00, A 0, B 0, C 0} C_DIS
LIN {X 93.49, Y 245.11, Z 0.00, A 0, B 0, C 0} C_DIS
LIN {X 93.69, Y 245.23, Z 0.00, A 0, B 0, C 0} C_DIS
LIN {X 93.88, Y 245.39, Z 0.00, A 0, B 0, C 0} C_DIS
LIN {X 94.06, Y 245.56, Z 0.00, A 0, B 0, C 0} C_DIS
LIN {X 94.26, Y 245.70, Z 0.00, A 0, B 0, C 0} C_DIS
LIN {X 94.46, Y 245.82, Z 0.00, A 0, B 0, C 0} C_DIS
LIN {X 94.65, Y 245.97, Z 0.00, A 0, B 0, C 0} C_DIS
LIN {X 94.84, Y 246.14, Z 0.00, A 0, B 0, C 0} C_DIS
LIN {X 95.03, Y 246.29, Z 0.00, A 0, B 0, C 0} C_DIS
LIN {X 95.23, Y 246.42, Z 0.00, A 0, B 0, C 0} C_DIS
LIN {X 95.43, Y 246.55, Z 0.00, A 0, B 0, C 0} C_DIS
LIN {X 95.62, Y 246.71, Z 0.00, A 0, B 0, C 0} C_DIS
LIN {X 95.81, Y 246.87, Z 0.00, A 0, B 0, C 0} C_DIS
LIN {X 96.00, Y 247.02, Z 0.00, A 0, B 0, C 0} C_DIS
LIN {X 96.21, Y 247.11, Z 0.00, A 0, B 0, C 0} C_DIS
LIN {X 96.42, Y 247.19, Z 0.00, A 0, B 0, C 0} C_DIS
LIN {X 96.62, Y 247.31, Z 0.00, A 0, B 0, C 0} C_DIS
LIN {X 96.82, Y 247.45, Z 0.00, A 0, B 0, C 0} C_DIS
LIN {X 97.02, Y 247.57, Z 0.00, A 0, B 0, C 0} C_DIS
LIN {X 97.23, Y 247.66, Z 0.00, A 0, B 0, C 0} C_DIS
LIN {X 97.44, Y 247.75, Z 0.00, A 0, B 0, C 0} C_DIS
LIN {X 97.64, Y 247.88, Z 0.00, A 0, B 0, C 0} C_DIS
LIN {X 97.82, Y 248.05, Z 0.00, A 0, B 0, C 0} C_DIS
LIN {X 98.01, Y 248.21, Z 0.00, A 0, B 0, C 0} C_DIS
LIN {X 98.21, Y 248.35, Z 0.00, A 0, B 0, C 0} C_DIS
LIN {X 98.41, Y 248.47, Z 0.00, A 0, B 0, C 0} C_DIS
LIN {X 98.60, Y 248.62, Z 0.00, A 0, B 0, C 0} C_DIS
LIN {X 98.79, Y 248.78, Z 0.00, A 0, B 0, C 0} C_DIS
LIN {X 98.98, Y 248.93, Z 0.00, A 0, B 0, C 0} C_DIS
LIN {X 99.18, Y 249.07, Z 0.00, A 0, B 0, C 0} C_DIS
LIN {X 99.38, Y 249.21, Z 0.00, A 0, B 0, C 0} C_DIS
LIN {X 99.57, Y 249.37, Z 0.00, A 0, B 0, C 0} C_DIS
LIN {X 99.75, Y 249.54, Z 0.00, A 0, B 0, C 0} C_DIS
LIN {X 99.93, Y 249.72, Z 0.00, A 0, B 0, C 0} C_DIS
LIN {X 100.11, Y 249.90, Z 0.00, A 0, B 0, C 0} C_DIS
LIN {X 100.29, Y 250.09, Z 0.00, A 0, B 0, C 0} C_DIS
LIN {X 100.47, Y 250.28, Z 0.00, A 0, B 0, C 0} C_DIS
LIN {X 100.65, Y 250.46, Z 0.00, A 0, B 0, C 0} C_DIS
LIN {X 100.83, Y 250.64, Z 0.00, A 0, B 0, C 0} C_DIS
LIN {X 101.02, Y 250.82, Z 0.00, A 0, B 0, C 0} C_DIS
LIN {X 101.20, Y 251.00, Z 0.00, A 0, B 0, C 0} C_DIS
LIN {X 101.38, Y 251.18, Z 0.00, A 0, B 0, C 0} C_DIS
LIN {X 101.55, Y 251.38, Z 0.00, A 0, B 0, C 0} C_DIS
LIN {X 101.71, Y 251.61, Z 0.00, A 0, B 0, C 0} C_DIS
LIN {X 101.86, Y 251.84, Z 0.00, A 0, B 0, C 0} C_DIS
LIN {X 102.02, Y 252.06, Z 0.00, A 0, B 0, C 0} C_DIS
LIN {X 102.20, Y 252.24, Z 0.00, A 0, B 0, C 0} C_DIS
LIN {X 102.38, Y 252.42, Z 0.00, A 0, B 0, C 0} C_DIS
LIN {X 102.57, Y 252.60, Z 0.00, A 0, B 0, C 0} C_DIS
LIN {X 102.75, Y 252.77, Z 0.00, A 0, B 0, C 0} C_DIS
LIN {X 102.93, Y 252.95, Z 0.00, A 0, B 0, C 0} C_DIS
LIN {X 103.11, Y 253.14, Z 0.00, A 0, B 0, C 0} C_DIS
LIN {X 103.28, Y 253.35, Z 0.00, A 0, B 0, C 0} C_DIS
LIN {X 103.44, Y 253.56, Z 0.00, A 0, B 0, C 0} C_DIS
LIN {X 103.59, Y 253.79, Z 0.00, A 0, B 0, C 0} C_DIS
LIN {X 103.74, Y 254.03, Z 0.00, A 0, B 0, C 0} C_DIS
LIN {X 103.90, Y 254.27, Z 0.00, A 0, B 0, C 0} C_DIS
LIN {X 104.05, Y 254.50, Z 0.00, A 0, B 0, C 0} C_DIS
LIN {X 104.20, Y 254.73, Z 0.00, A 0, B 0, C 0} C_DIS
LIN {X 104.35, Y 254.98, Z 0.00, A 0, B 0, C 0} C_DIS
LIN {X 104.47, Y 255.24, Z 0.00, A 0, B 0, C 0} C_DIS
LIN {X 104.59, Y 255.51, Z 0.00, A 0, B 0, C 0} C_DIS
LIN {X 104.71, Y 255.79, Z 0.00, A 0, B 0, C 0} C_DIS
LIN {X 104.83, Y 256.07, Z 0.00, A 0, B 0, C 0} C_DIS
LIN {X 104.95, Y 256.34, Z 0.00, A 0, B 0, C 0} C_DIS
LIN {X 105.07, Y 256.62, Z 0.00, A 0, B 0, C 0} C_DIS
LIN {X 105.19, Y 256.89, Z 0.00, A 0, B 0, C 0} C_DIS
LIN {X 105.31, Y 257.15, Z 0.00, A 0, B 0, C 0} C_DIS
LIN {X 105.44, Y 257.42, Z 0.00, A 0, B 0, C 0} C_DIS
LIN {X 105.56, Y 257.68, Z 0.00, A 0, B 0, C 0} C_DIS
LIN {X 105.68, Y 257.97, Z 0.00, A 0, B 0, C 0} C_DIS
LIN {X 105.77, Y 258.29, Z 0.00, A 0, B 0, C 0} C_DIS
LIN {X 105.78, Y 258.60, Z 0.00, A 0, B 0, C 0} C_DIS
LIN {X 105.67, Y 258.82, Z 0.00, A 0, B 0, C 0} C_DIS
LIN {X 105.47, Y 258.85, Z 0.00, A 0, B 0, C 0} C_DIS
LIN {X 105.24, Y 258.76, Z 0.00, A 0, B 0, C 0} C_DIS
LIN {X 105.02, Y 258.67, Z 0.00, A 0, B 0, C 0} C_DIS
LIN {X 104.82, Y 258.59, Z 0.00, A 0, B 0, C 0} C_DIS
LIN {X 104.61, Y 258.51, Z 0.00, A 0, B 0, C 0} C_DIS
LIN {X 104.39, Y 258.46, Z 0.00, A 0, B 0, C 0} C_DIS
LIN {X 104.18, Y 258.42, Z 0.00, A 0, B 0, C 0} C_DIS
LIN {X 103.96, Y 258.40, Z 0.00, A 0, B 0, C 0} C_DIS
LIN {X 103.74, Y 258.40, Z 0.00, A 0, B 0, C 0} C_DIS
LIN {X 103.53, Y 258.40, Z 0.00, A 0, B 0, C 0} C_DIS
LIN {X 103.31, Y 258.41, Z 0.00, A 0, B 0, C 0} C_DIS
LIN {X 103.09, Y 258.41, Z 0.00, A 0, B 0, C 0} C_DIS
LIN {X 102.87, Y 258.41, Z 0.00, A 0, B 0, C 0} C_DIS
LIN {X 102.66, Y 258.41, Z 0.00, A 0, B 0, C 0} C_DIS
LIN {X 102.44, Y 258.41, Z 0.00, A 0, B 0, C 0} C_DIS
LIN {X 102.22, Y 258.41, Z 0.00, A 0, B 0, C 0} C_DIS
LIN {X 102.00, Y 258.41, Z 0.00, A 0, B 0, C 0} C_DIS
LIN {X 101.79, Y 258.41, Z 0.00, A 0, B 0, C 0} C_DIS
LIN {X 101.57, Y 258.41, Z 0.00, A 0, B 0, C 0} C_DIS
LIN {X 101.35, Y 258.41, Z 0.00, A 0, B 0, C 0} C_DIS
LIN {X 101.13, Y 258.41, Z 0.00, A 0, B 0, C 0} C_DIS
LIN {X 100.92, Y 258.41, Z 0.00, A 0, B 0, C 0} C_DIS
LIN {X 100.70, Y 258.41, Z 0.00, A 0, B 0, C 0} C_DIS
LIN {X 100.48, Y 258.41, Z 0.00, A 0, B 0, C 0} C_DIS
LIN {X 100.26, Y 258.41, Z 0.00, A 0, B 0, C 0} C_DIS
LIN {X 100.05, Y 258.41, Z 0.00, A 0, B 0, C 0} C_DIS
LIN {X 99.83, Y 258.41, Z 0.00, A 0, B 0, C 0} C_DIS
LIN {X 99.61, Y 258.41, Z 0.00, A 0, B 0, C 0} C_DIS
LIN {X 99.40, Y 258.41, Z 0.00, A 0, B 0, C 0} C_DIS
LIN {X 99.18, Y 258.41, Z 0.00, A 0, B 0, C 0} C_DIS
LIN {X 98.96, Y 258.41, Z 0.00, A 0, B 0, C 0} C_DIS
LIN {X 98.74, Y 258.41, Z 0.00, A 0, B 0, C 0} C_DIS
LIN {X 98.53, Y 258.41, Z 0.00, A 0, B 0, C 0} C_DIS
LIN {X 98.31, Y 258.41, Z 0.00, A 0, B 0, C 0} C_DIS
LIN {X 98.09, Y 258.41, Z 0.00, A 0, B 0, C 0} C_DIS
LIN {X 97.87, Y 258.41, Z 0.00, A 0, B 0, C 0} C_DIS
LIN {X 97.66, Y 258.41, Z 0.00, A 0, B 0, C 0} C_DIS
LIN {X 97.44, Y 258.41, Z 0.00, A 0, B 0, C 0} C_DIS
LIN {X 97.22, Y 258.41, Z 0.00, A 0, B 0, C 0} C_DIS
LIN {X 97.00, Y 258.41, Z 0.00, A 0, B 0, C 0} C_DIS
LIN {X 96.79, Y 258.41, Z 0.00, A 0, B 0, C 0} C_DIS
LIN {X 96.57, Y 258.41, Z 0.00, A 0, B 0, C 0} C_DIS
LIN {X 96.35, Y 258.41, Z 0.00, A 0, B 0, C 0} C_DIS
LIN {X 96.13, Y 258.41, Z 0.00, A 0, B 0, C 0} C_DIS
LIN {X 95.92, Y 258.41, Z 0.00, A 0, B 0, C 0} C_DIS
LIN {X 95.70, Y 258.41, Z 0.00, A 0, B 0, C 0} C_DIS
LIN {X 95.48, Y 258.41, Z 0.00, A 0, B 0, C 0} C_DIS
LIN {X 95.26, Y 258.41, Z 0.00, A 0, B 0, C 0} C_DIS
LIN {X 95.05, Y 258.41, Z 0.00, A 0, B 0, C 0} C_DIS
LIN {X 94.83, Y 258.41, Z 0.00, A 0, B 0, C 0} C_DIS
LIN {X 94.61, Y 258.41, Z 0.00, A 0, B 0, C 0} C_DIS
LIN {X 94.39, Y 258.41, Z 0.00, A 0, B 0, C 0} C_DIS
LIN {X 94.18, Y 258.41, Z 0.00, A 0, B 0, C 0} C_DIS
LIN {X 93.96, Y 258.41, Z 0.00, A 0, B 0, C 0} C_DIS
LIN {X 93.74, Y 258.41, Z 0.00, A 0, B 0, C 0} C_DIS
LIN {X 93.52, Y 258.41, Z 0.00, A 0, B 0, C 0} C_DIS
LIN {X 93.31, Y 258.41, Z 0.00, A 0, B 0, C 0} C_DIS
LIN {X 93.09, Y 258.41, Z 0.00, A 0, B 0, C 0} C_DIS
LIN {X 92.87, Y 258.41, Z 0.00, A 0, B 0, C 0} C_DIS
LIN {X 92.65, Y 258.41, Z 0.00, A 0, B 0, C 0} C_DIS
LIN {X 92.44, Y 258.41, Z 0.00, A 0, B 0, C 0} C_DIS
LIN {X 92.22, Y 258.41, Z 0.00, A 0, B 0, C 0} C_DIS
LIN {X 92.00, Y 258.41, Z 0.00, A 0, B 0, C 0} C_DIS
LIN {X 91.78, Y 258.41, Z 0.00, A 0, B 0, C 0} C_DIS
LIN {X 91.57, Y 258.41, Z 0.00, A 0, B 0, C 0} C_DIS
LIN {X 91.35, Y 258.41, Z 0.00, A 0, B 0, C 0} C_DIS
LIN {X 91.13, Y 258.41, Z 0.00, A 0, B 0, C 0} C_DIS
LIN {X 90.91, Y 258.41, Z 0.00, A 0, B 0, C 0} C_DIS
LIN {X 90.70, Y 258.41, Z 0.00, A 0, B 0, C 0} C_DIS
LIN {X 90.48, Y 258.41, Z 0.00, A 0, B 0, C 0} C_DIS
LIN {X 90.26, Y 258.41, Z 0.00, A 0, B 0, C 0} C_DIS
LIN {X 90.05, Y 258.41, Z 0.00, A 0, B 0, C 0} C_DIS
LIN {X 89.83, Y 258.41, Z 0.00, A 0, B 0, C 0} C_DIS
LIN {X 89.61, Y 258.41, Z 0.00, A 0, B 0, C 0} C_DIS
LIN {X 89.39, Y 258.41, Z 0.00, A 0, B 0, C 0} C_DIS
LIN {X 89.18, Y 258.41, Z 0.00, A 0, B 0, C 0} C_DIS
LIN {X 88.96, Y 258.41, Z 0.00, A 0, B 0, C 0} C_DIS
LIN {X 88.74, Y 258.41, Z 0.00, A 0, B 0, C 0} C_DIS
LIN {X 88.52, Y 258.41, Z 0.00, A 0, B 0, C 0} C_DIS
LIN {X 88.31, Y 258.41, Z 0.00, A 0, B 0, C 0} C_DIS
LIN {X 88.09, Y 258.41, Z 0.00, A 0, B 0, C 0} C_DIS
LIN {X 87.87, Y 258.41, Z 0.00, A 0, B 0, C 0} C_DIS
LIN {X 87.65, Y 258.41, Z 0.00, A 0, B 0, C 0} C_DIS
LIN {X 87.44, Y 258.41, Z 0.00, A 0, B 0, C 0} C_DIS
LIN {X 87.22, Y 258.41, Z 0.00, A 0, B 0, C 0} C_DIS
LIN {X 87.00, Y 258.41, Z 0.00, A 0, B 0, C 0} C_DIS
LIN {X 86.78, Y 258.41, Z 0.00, A 0, B 0, C 0} C_DIS
LIN {X 86.57, Y 258.41, Z 0.00, A 0, B 0, C 0} C_DIS
LIN {X 86.35, Y 258.41, Z 0.00, A 0, B 0, C 0} C_DIS
LIN {X 86.13, Y 258.41, Z 0.00, A 0, B 0, C 0} C_DIS
LIN {X 85.91, Y 258.41, Z 0.00, A 0, B 0, C 0} C_DIS
LIN {X 85.70, Y 258.41, Z 0.00, A 0, B 0, C 0} C_DIS
LIN {X 85.48, Y 258.41, Z 0.00, A 0, B 0, C 0} C_DIS
LIN {X 85.26, Y 258.41, Z 0.00, A 0, B 0, C 0} C_DIS
LIN {X 85.04, Y 258.41, Z 0.00, A 0, B 0, C 0} C_DIS
LIN {X 84.83, Y 258.41, Z 0.00, A 0, B 0, C 0} C_DIS
LIN {X 84.61, Y 258.41, Z 0.00, A 0, B 0, C 0} C_DIS
LIN {X 84.39, Y 258.41, Z 0.00, A 0, B 0, C 0} C_DIS
LIN {X 84.17, Y 258.41, Z 0.00, A 0, B 0, C 0} C_DIS
LIN {X 83.96, Y 258.41, Z 0.00, A 0, B 0, C 0} C_DIS
LIN {X 83.74, Y 258.41, Z 0.00, A 0, B 0, C 0} C_DIS
LIN {X 83.52, Y 258.41, Z 0.00, A 0, B 0, C 0} C_DIS
LIN {X 83.30, Y 258.41, Z 0.00, A 0, B 0, C 0} C_DIS
LIN {X 83.09, Y 258.41, Z 0.00, A 0, B 0, C 0} C_DIS
LIN {X 82.87, Y 258.41, Z 0.00, A 0, B 0, C 0} C_DIS
LIN {X 82.65, Y 258.41, Z 0.00, A 0, B 0, C 0} C_DIS
LIN {X 82.43, Y 258.41, Z 0.00, A 0, B 0, C 0} C_DIS
LIN {X 82.22, Y 258.41, Z 0.00, A 0, B 0, C 0} C_DIS
LIN {X 82.00, Y 258.41, Z 0.00, A 0, B 0, C 0} C_DIS
LIN {X 81.78, Y 258.41, Z 0.00, A 0, B 0, C 0} C_DIS
LIN {X 81.57, Y 258.41, Z 0.00, A 0, B 0, C 0} C_DIS
LIN {X 81.35, Y 258.41, Z 0.00, A 0, B 0, C 0} C_DIS
LIN {X 81.13, Y 258.41, Z 0.00, A 0, B 0, C 0} C_DIS
LIN {X 80.91, Y 258.41, Z 0.00, A 0, B 0, C 0} C_DIS
LIN {X 80.70, Y 258.41, Z 0.00, A 0, B 0, C 0} C_DIS
LIN {X 80.48, Y 258.41, Z 0.00, A 0, B 0, C 0} C_DIS
LIN {X 80.26, Y 258.41, Z 0.00, A 0, B 0, C 0} C_DIS
LIN {X 80.04, Y 258.41, Z 0.00, A 0, B 0, C 0} C_DIS
LIN {X 79.83, Y 258.41, Z 0.00, A 0, B 0, C 0} C_DIS
LIN {X 79.61, Y 258.41, Z 0.00, A 0, B 0, C 0} C_DIS
LIN {X 79.39, Y 258.41, Z 0.00, A 0, B 0, C 0} C_DIS
LIN {X 79.17, Y 258.41, Z 0.00, A 0, B 0, C 0} C_DIS
LIN {X 78.96, Y 258.41, Z 0.00, A 0, B 0, C 0} C_DIS
LIN {X 78.74, Y 258.41, Z 0.00, A 0, B 0, C 0} C_DIS
LIN {X 78.52, Y 258.41, Z 0.00, A 0, B 0, C 0} C_DIS
LIN {X 78.30, Y 258.41, Z 0.00, A 0, B 0, C 0} C_DIS
LIN {X 78.09, Y 258.41, Z 0.00, A 0, B 0, C 0} C_DIS
LIN {X 77.87, Y 258.41, Z 0.00, A 0, B 0, C 0} C_DIS
LIN {X 77.65, Y 258.41, Z 0.00, A 0, B 0, C 0} C_DIS
LIN {X 77.43, Y 258.41, Z 0.00, A 0, B 0, C 0} C_DIS
LIN {X 77.22, Y 258.41, Z 0.00, A 0, B 0, C 0} C_DIS
LIN {X 77.00, Y 258.41, Z 0.00, A 0, B 0, C 0} C_DIS
LIN {X 76.78, Y 258.41, Z 0.00, A 0, B 0, C 0} C_DIS
LIN {X 76.56, Y 258.41, Z 0.00, A 0, B 0, C 0} C_DIS
LIN {X 76.35, Y 258.41, Z 0.00, A 0, B 0, C 0} C_DIS
LIN {X 76.13, Y 258.41, Z 0.00, A 0, B 0, C 0} C_DIS
LIN {X 75.91, Y 258.41, Z 0.00, A 0, B 0, C 0} C_DIS
LIN {X 75.69, Y 258.41, Z 0.00, A 0, B 0, C 0} C_DIS
LIN {X 75.48, Y 258.41, Z 0.00, A 0, B 0, C 0} C_DIS
LIN {X 75.26, Y 258.41, Z 0.00, A 0, B 0, C 0} C_DIS
LIN {X 75.04, Y 258.41, Z 0.00, A 0, B 0, C 0} C_DIS
LIN {X 74.82, Y 258.41, Z 0.00, A 0, B 0, C 0} C_DIS
LIN {X 74.61, Y 258.41, Z 0.00, A 0, B 0, C 0} C_DIS
LIN {X 74.39, Y 258.41, Z 0.00, A 0, B 0, C 0} C_DIS
LIN {X 74.17, Y 258.41, Z 0.00, A 0, B 0, C 0} C_DIS
LIN {X 73.95, Y 258.41, Z 0.00, A 0, B 0, C 0} C_DIS
LIN {X 73.74, Y 258.41, Z 0.00, A 0, B 0, C 0} C_DIS
LIN {X 73.52, Y 258.41, Z 0.00, A 0, B 0, C 0} C_DIS
LIN {X 73.30, Y 258.41, Z 0.00, A 0, B 0, C 0} C_DIS
LIN {X 73.08, Y 258.41, Z 0.00, A 0, B 0, C 0} C_DIS
LIN {X 72.87, Y 258.41, Z 0.00, A 0, B 0, C 0} C_DIS
LIN {X 72.65, Y 258.41, Z 0.00, A 0, B 0, C 0} C_DIS
LIN {X 72.43, Y 258.41, Z 0.00, A 0, B 0, C 0} C_DIS
LIN {X 72.22, Y 258.41, Z 0.00, A 0, B 0, C 0} C_DIS
LIN {X 72.00, Y 258.41, Z 0.00, A 0, B 0, C 0} C_DIS
LIN {X 71.78, Y 258.41, Z 0.00, A 0, B 0, C 0} C_DIS
LIN {X 71.56, Y 258.41, Z 0.00, A 0, B 0, C 0} C_DIS
LIN {X 71.35, Y 258.41, Z 0.00, A 0, B 0, C 0} C_DIS
LIN {X 71.13, Y 258.41, Z 0.00, A 0, B 0, C 0} C_DIS
LIN {X 70.91, Y 258.41, Z 0.00, A 0, B 0, C 0} C_DIS
LIN {X 70.69, Y 258.41, Z 0.00, A 0, B 0, C 0} C_DIS
LIN {X 70.48, Y 258.41, Z 0.00, A 0, B 0, C 0} C_DIS
LIN {X 70.26, Y 258.41, Z 0.00, A 0, B 0, C 0} C_DIS
LIN {X 70.04, Y 258.41, Z 0.00, A 0, B 0, C 0} C_DIS
LIN {X 69.82, Y 258.41, Z 0.00, A 0, B 0, C 0} C_DIS
LIN {X 69.61, Y 258.41, Z 0.00, A 0, B 0, C 0} C_DIS
LIN {X 69.39, Y 258.41, Z 0.00, A 0, B 0, C 0} C_DIS
LIN {X 69.17, Y 258.41, Z 0.00, A 0, B 0, C 0} C_DIS
LIN {X 68.95, Y 258.41, Z 0.00, A 0, B 0, C 0} C_DIS
LIN {X 68.74, Y 258.41, Z 0.00, A 0, B 0, C 0} C_DIS
LIN {X 68.52, Y 258.41, Z 0.00, A 0, B 0, C 0} C_DIS
LIN {X 68.30, Y 258.40, Z 0.00, A 0, B 0, C 0} C_DIS
LIN {X 68.08, Y 258.40, Z 0.00, A 0, B 0, C 0} C_DIS
LIN {X 67.87, Y 258.40, Z 0.00, A 0, B 0, C 0} C_DIS
LIN {X 67.65, Y 258.40, Z 0.00, A 0, B 0, C 0} C_DIS
LIN {X 67.43, Y 258.40, Z 0.00, A 0, B 0, C 0} C_DIS
LIN {X 67.21, Y 258.40, Z 0.00, A 0, B 0, C 0} C_DIS
LIN {X 67.00, Y 258.40, Z 0.00, A 0, B 0, C 0} C_DIS
LIN {X 66.78, Y 258.40, Z 0.00, A 0, B 0, C 0} C_DIS
LIN {X 66.56, Y 258.40, Z 0.00, A 0, B 0, C 0} C_DIS
LIN {X 66.34, Y 258.40, Z 0.00, A 0, B 0, C 0} C_DIS
LIN {X 66.13, Y 258.40, Z 0.00, A 0, B 0, C 0} C_DIS
LIN {X 65.91, Y 258.40, Z 0.00, A 0, B 0, C 0} C_DIS
LIN {X 65.69, Y 258.40, Z 0.00, A 0, B 0, C 0} C_DIS
LIN {X 65.48, Y 258.40, Z 0.00, A 0, B 0, C 0} C_DIS
LIN {X 65.26, Y 258.40, Z 0.00, A 0, B 0, C 0} C_DIS
LIN {X 65.04, Y 258.40, Z 0.00, A 0, B 0, C 0} C_DIS
LIN {X 64.82, Y 258.41, Z 0.00, A 0, B 0, C 0} C_DIS
LIN {X 64.61, Y 258.41, Z 0.00, A 0, B 0, C 0} C_DIS
LIN {X 64.39, Y 258.41, Z 0.00, A 0, B 0, C 0} C_DIS
LIN {X 64.17, Y 258.41, Z 0.00, A 0, B 0, C 0} C_DIS
LIN {X 63.95, Y 258.41, Z 0.00, A 0, B 0, C 0} C_DIS
LIN {X 63.74, Y 258.41, Z 0.00, A 0, B 0, C 0} C_DIS
LIN {X 63.52, Y 258.41, Z 0.00, A 0, B 0, C 0} C_DIS
LIN {X 63.30, Y 258.41, Z 0.00, A 0, B 0, C 0} C_DIS
LIN {X 63.08, Y 258.41, Z 0.00, A 0, B 0, C 0} C_DIS
LIN {X 62.86, Y 258.41, Z 0.00, A 0, B 0, C 0} C_DIS
LIN {X 62.65, Y 258.42, Z 0.00, A 0, B 0, C 0} C_DIS
LIN {X 62.43, Y 258.42, Z 0.00, A 0, B 0, C 0} C_DIS
LIN {X 62.21, Y 258.42, Z 0.00, A 0, B 0, C 0} C_DIS
LIN {X 61.99, Y 258.42, Z 0.00, A 0, B 0, C 0} C_DIS
LIN {X 61.78, Y 258.41, Z 0.00, A 0, B 0, C 0} C_DIS
LIN {X 61.56, Y 258.40, Z 0.00, A 0, B 0, C 0} C_DIS
LIN {X 61.35, Y 258.37, Z 0.00, A 0, B 0, C 0} C_DIS
LIN {X 61.13, Y 258.33, Z 0.00, A 0, B 0, C 0} C_DIS
LIN {X 60.92, Y 258.28, Z 0.00, A 0, B 0, C 0} C_DIS
LIN {X 60.71, Y 258.21, Z 0.00, A 0, B 0, C 0} C_DIS
LIN {X 60.49, Y 258.13, Z 0.00, A 0, B 0, C 0} C_DIS
LIN {X 60.28, Y 258.04, Z 0.00, A 0, B 0, C 0} C_DIS
LIN {X 60.07, Y 257.96, Z 0.00, A 0, B 0, C 0} C_DIS
LIN {X 59.86, Y 257.89, Z 0.00, A 0, B 0, C 0} C_DIS
LIN {X 59.65, Y 257.82, Z 0.00, A 0, B 0, C 0} C_DIS
LIN {X 59.43, Y 257.77, Z 0.00, A 0, B 0, C 0} C_DIS
LIN {X 59.22, Y 257.73, Z 0.00, A 0, B 0, C 0} C_DIS
LIN {X 59.00, Y 257.68, Z 0.00, A 0, B 0, C 0} C_DIS
LIN {X 58.79, Y 257.63, Z 0.00, A 0, B 0, C 0} C_DIS
LIN {X 58.58, Y 257.57, Z 0.00, A 0, B 0, C 0} C_DIS
LIN {X 58.36, Y 257.50, Z 0.00, A 0, B 0, C 0} C_DIS
LIN {X 58.15, Y 257.42, Z 0.00, A 0, B 0, C 0} C_DIS
LIN {X 57.94, Y 257.34, Z 0.00, A 0, B 0, C 0} C_DIS
LIN {X 57.73, Y 257.25, Z 0.00, A 0, B 0, C 0} C_DIS
LIN {X 57.52, Y 257.17, Z 0.00, A 0, B 0, C 0} C_DIS
LIN {X 57.31, Y 257.08, Z 0.00, A 0, B 0, C 0} C_DIS
LIN {X 57.10, Y 257.00, Z 0.00, A 0, B 0, C 0} C_DIS
LIN {X 56.89, Y 256.92, Z 0.00, A 0, B 0, C 0} C_DIS
LIN {X 56.68, Y 256.84, Z 0.00, A 0, B 0, C 0} C_DIS
LIN {X 56.47, Y 256.76, Z 0.00, A 0, B 0, C 0} C_DIS
LIN {X 56.26, Y 256.69, Z 0.00, A 0, B 0, C 0} C_DIS
LIN {X 56.05, Y 256.61, Z 0.00, A 0, B 0, C 0} C_DIS
LIN {X 55.83, Y 256.53, Z 0.00, A 0, B 0, C 0} C_DIS
LIN {X 55.62, Y 256.46, Z 0.00, A 0, B 0, C 0} C_DIS
LIN {X 55.41, Y 256.38, Z 0.00, A 0, B 0, C 0} C_DIS
LIN {X 55.20, Y 256.30, Z 0.00, A 0, B 0, C 0} C_DIS
LIN {X 54.99, Y 256.21, Z 0.00, A 0, B 0, C 0} C_DIS
LIN {X 54.78, Y 256.12, Z 0.00, A 0, B 0, C 0} C_DIS
LIN {X 54.58, Y 256.01, Z 0.00, A 0, B 0, C 0} C_DIS
LIN {X 54.39, Y 255.86, Z 0.00, A 0, B 0, C 0} C_DIS
LIN {X 54.20, Y 255.68, Z 0.00, A 0, B 0, C 0} C_DIS
LIN {X 54.01, Y 255.53, Z 0.00, A 0, B 0, C 0} C_DIS
LIN {X 53.80, Y 255.43, Z 0.00, A 0, B 0, C 0} C_DIS
LIN {X 53.59, Y 255.35, Z 0.00, A 0, B 0, C 0} C_DIS
LIN {X 53.39, Y 255.24, Z 0.00, A 0, B 0, C 0} C_DIS
LIN {X 53.19, Y 255.11, Z 0.00, A 0, B 0, C 0} C_DIS
LIN {X 52.99, Y 254.98, Z 0.00, A 0, B 0, C 0} C_DIS
LIN {X 52.78, Y 254.88, Z 0.00, A 0, B 0, C 0} C_DIS
LIN {X 52.57, Y 254.79, Z 0.00, A 0, B 0, C 0} C_DIS
LIN {X 52.37, Y 254.68, Z 0.00, A 0, B 0, C 0} C_DIS
LIN {X 52.18, Y 254.52, Z 0.00, A 0, B 0, C 0} C_DIS
LIN {X 52.00, Y 254.35, Z 0.00, A 0, B 0, C 0} C_DIS
LIN {X 51.80, Y 254.21, Z 0.00, A 0, B 0, C 0} C_DIS
LIN {X 51.60, Y 254.08, Z 0.00, A 0, B 0, C 0} C_DIS
LIN {X 51.40, Y 253.94, Z 0.00, A 0, B 0, C 0} C_DIS
LIN {X 51.22, Y 253.78, Z 0.00, A 0, B 0, C 0} C_DIS
LIN {X 51.03, Y 253.62, Z 0.00, A 0, B 0, C 0} C_DIS
LIN {X 50.83, Y 253.49, Z 0.00, A 0, B 0, C 0} C_DIS
LIN {X 50.63, Y 253.35, Z 0.00, A 0, B 0, C 0} C_DIS
LIN {X 50.44, Y 253.21, Z 0.00, A 0, B 0, C 0} C_DIS
LIN {X 50.25, Y 253.05, Z 0.00, A 0, B 0, C 0} C_DIS
LIN {X 50.06, Y 252.90, Z 0.00, A 0, B 0, C 0} C_DIS
LIN {X 49.86, Y 252.76, Z 0.00, A 0, B 0, C 0} C_DIS
LIN {X 49.66, Y 252.63, Z 0.00, A 0, B 0, C 0} C_DIS
LIN {X 49.47, Y 252.46, Z 0.00, A 0, B 0, C 0} C_DIS
LIN {X 49.28, Y 252.31, Z 0.00, A 0, B 0, C 0} C_DIS
LIN {X 49.08, Y 252.18, Z 0.00, A 0, B 0, C 0} C_DIS
LIN {X 48.89, Y 252.04, Z 0.00, A 0, B 0, C 0} C_DIS
LIN {X 48.70, Y 251.88, Z 0.00, A 0, B 0, C 0} C_DIS
LIN {X 48.51, Y 251.71, Z 0.00, A 0, B 0, C 0} C_DIS
LIN {X 48.33, Y 251.53, Z 0.00, A 0, B 0, C 0} C_DIS
LIN {X 48.15, Y 251.35, Z 0.00, A 0, B 0, C 0} C_DIS
LIN {X 47.97, Y 251.16, Z 0.00, A 0, B 0, C 0} C_DIS
LIN {X 47.79, Y 250.98, Z 0.00, A 0, B 0, C 0} C_DIS
LIN {X 47.61, Y 250.79, Z 0.00, A 0, B 0, C 0} C_DIS
LIN {X 47.43, Y 250.61, Z 0.00, A 0, B 0, C 0} C_DIS
LIN {X 47.25, Y 250.43, Z 0.00, A 0, B 0, C 0} C_DIS
LIN {X 47.07, Y 250.25, Z 0.00, A 0, B 0, C 0} C_DIS
LIN {X 46.89, Y 250.07, Z 0.00, A 0, B 0, C 0} C_DIS
LIN {X 46.70, Y 249.89, Z 0.00, A 0, B 0, C 0} C_DIS
LIN {X 46.52, Y 249.71, Z 0.00, A 0, B 0, C 0} C_DIS
LIN {X 46.34, Y 249.53, Z 0.00, A 0, B 0, C 0} C_DIS
LIN {X 46.16, Y 249.35, Z 0.00, A 0, B 0, C 0} C_DIS
LIN {X 45.98, Y 249.16, Z 0.00, A 0, B 0, C 0} C_DIS
LIN {X 45.80, Y 248.98, Z 0.00, A 0, B 0, C 0} C_DIS
LIN {X 45.62, Y 248.79, Z 0.00, A 0, B 0, C 0} C_DIS
LIN {X 45.45, Y 248.60, Z 0.00, A 0, B 0, C 0} C_DIS
LIN {X 45.28, Y 248.40, Z 0.00, A 0, B 0, C 0} C_DIS
LIN {X 45.12, Y 248.17, Z 0.00, A 0, B 0, C 0} C_DIS
LIN {X 44.97, Y 247.93, Z 0.00, A 0, B 0, C 0} C_DIS
LIN {X 44.83, Y 247.69, Z 0.00, A 0, B 0, C 0} C_DIS
LIN {X 44.67, Y 247.46, Z 0.00, A 0, B 0, C 0} C_DIS
LIN {X 44.51, Y 247.25, Z 0.00, A 0, B 0, C 0} C_DIS
LIN {X 44.33, Y 247.05, Z 0.00, A 0, B 0, C 0} C_DIS
LIN {X 44.15, Y 246.87, Z 0.00, A 0, B 0, C 0} C_DIS
LIN {X 43.96, Y 246.70, Z 0.00, A 0, B 0, C 0} C_DIS
LIN {X 43.78, Y 246.53, Z 0.00, A 0, B 0, C 0} C_DIS
LIN {X 43.59, Y 246.35, Z 0.00, A 0, B 0, C 0} C_DIS
LIN {X 43.42, Y 246.16, Z 0.00, A 0, B 0, C 0} C_DIS
LIN {X 43.25, Y 245.95, Z 0.00, A 0, B 0, C 0} C_DIS
LIN {X 43.09, Y 245.73, Z 0.00, A 0, B 0, C 0} C_DIS
LIN {X 42.93, Y 245.51, Z 0.00, A 0, B 0, C 0} C_DIS
LIN {X 42.78, Y 245.28, Z 0.00, A 0, B 0, C 0} C_DIS
LIN {X 42.63, Y 245.04, Z 0.00, A 0, B 0, C 0} C_DIS
LIN {X 42.48, Y 244.81, Z 0.00, A 0, B 0, C 0} C_DIS
LIN {X 42.32, Y 244.57, Z 0.00, A 0, B 0, C 0} C_DIS
LIN {X 42.17, Y 244.35, Z 0.00, A 0, B 0, C 0} C_DIS
LIN {X 42.01, Y 244.12, Z 0.00, A 0, B 0, C 0} C_DIS
LIN {X 41.85, Y 243.89, Z 0.00, A 0, B 0, C 0} C_DIS
LIN {X 41.70, Y 243.66, Z 0.00, A 0, B 0, C 0} C_DIS
LIN {X 41.55, Y 243.42, Z 0.00, A 0, B 0, C 0} C_DIS
LIN {X 41.40, Y 243.18, Z 0.00, A 0, B 0, C 0} C_DIS
LIN {X 41.26, Y 242.93, Z 0.00, A 0, B 0, C 0} C_DIS
LIN {X 41.13, Y 242.67, Z 0.00, A 0, B 0, C 0} C_DIS
LIN {X 41.01, Y 242.40, Z 0.00, A 0, B 0, C 0} C_DIS
LIN {X 40.89, Y 242.13, Z 0.00, A 0, B 0, C 0} C_DIS
LIN {X 40.77, Y 241.85, Z 0.00, A 0, B 0, C 0} C_DIS
LIN {X 40.66, Y 241.57, Z 0.00, A 0, B 0, C 0} C_DIS
LIN {X 40.54, Y 241.30, Z 0.00, A 0, B 0, C 0} C_DIS
LIN {X 40.40, Y 241.04, Z 0.00, A 0, B 0, C 0} C_DIS
LIN {X 40.26, Y 240.80, Z 0.00, A 0, B 0, C 0} C_DIS
LIN {X 40.10, Y 240.57, Z 0.00, A 0, B 0, C 0} C_DIS
LIN {X 39.94, Y 240.35, Z 0.00, A 0, B 0, C 0} C_DIS
LIN {X 39.78, Y 240.12, Z 0.00, A 0, B 0, C 0} C_DIS
LIN {X 39.64, Y 239.88, Z 0.00, A 0, B 0, C 0} C_DIS
LIN {X 39.50, Y 239.63, Z 0.00, A 0, B 0, C 0} C_DIS
LIN {X 39.38, Y 239.36, Z 0.00, A 0, B 0, C 0} C_DIS
LIN {X 39.26, Y 239.08, Z 0.00, A 0, B 0, C 0} C_DIS
LIN {X 39.14, Y 238.81, Z 0.00, A 0, B 0, C 0} C_DIS
LIN {X 39.02, Y 238.53, Z 0.00, A 0, B 0, C 0} C_DIS
LIN {X 38.90, Y 238.26, Z 0.00, A 0, B 0, C 0} C_DIS
LIN {X 38.77, Y 238.00, Z 0.00, A 0, B 0, C 0} C_DIS
LIN {X 38.63, Y 237.75, Z 0.00, A 0, B 0, C 0} C_DIS
LIN {X 38.49, Y 237.50, Z 0.00, A 0, B 0, C 0} C_DIS
LIN {X 38.35, Y 237.26, Z 0.00, A 0, B 0, C 0} C_DIS
LIN {X 38.21, Y 237.01, Z 0.00, A 0, B 0, C 0} C_DIS
LIN {X 38.07, Y 236.75, Z 0.00, A 0, B 0, C 0} C_DIS
LIN {X 37.95, Y 236.49, Z 0.00, A 0, B 0, C 0} C_DIS
LIN {X 37.83, Y 236.20, Z 0.00, A 0, B 0, C 0} C_DIS
LIN {X 37.73, Y 235.91, Z 0.00, A 0, B 0, C 0} C_DIS
LIN {X 37.64, Y 235.61, Z 0.00, A 0, B 0, C 0} C_DIS
LIN {X 37.55, Y 235.32, Z 0.00, A 0, B 0, C 0} C_DIS
LIN {X 37.45, Y 235.03, Z 0.00, A 0, B 0, C 0} C_DIS
LIN {X 37.34, Y 234.75, Z 0.00, A 0, B 0, C 0} C_DIS
LIN {X 37.23, Y 234.47, Z 0.00, A 0, B 0, C 0} C_DIS
LIN {X 37.11, Y 234.20, Z 0.00, A 0, B 0, C 0} C_DIS
LIN {X 36.98, Y 233.93, Z 0.00, A 0, B 0, C 0} C_DIS
LIN {X 36.86, Y 233.66, Z 0.00, A 0, B 0, C 0} C_DIS
LIN {X 36.73, Y 233.39, Z 0.00, A 0, B 0, C 0} C_DIS
LIN {X 36.61, Y 233.12, Z 0.00, A 0, B 0, C 0} C_DIS
LIN {X 36.50, Y 232.84, Z 0.00, A 0, B 0, C 0} C_DIS
LIN {X 36.40, Y 232.55, Z 0.00, A 0, B 0, C 0} C_DIS
LIN {X 36.30, Y 232.26, Z 0.00, A 0, B 0, C 0} C_DIS
LIN {X 36.22, Y 231.95, Z 0.00, A 0, B 0, C 0} C_DIS
LIN {X 36.12, Y 231.66, Z 0.00, A 0, B 0, C 0} C_DIS
LIN {X 36.01, Y 231.38, Z 0.00, A 0, B 0, C 0} C_DIS
LIN {X 35.91, Y 231.09, Z 0.00, A 0, B 0, C 0} C_DIS
LIN {X 35.83, Y 230.79, Z 0.00, A 0, B 0, C 0} C_DIS
LIN {X 35.74, Y 230.49, Z 0.00, A 0, B 0, C 0} C_DIS
LIN {X 35.63, Y 230.21, Z 0.00, A 0, B 0, C 0} C_DIS
LIN {X 35.52, Y 229.92, Z 0.00, A 0, B 0, C 0} C_DIS
LIN {X 35.44, Y 229.63, Z 0.00, A 0, B 0, C 0} C_DIS
LIN {X 35.38, Y 229.31, Z 0.00, A 0, B 0, C 0} C_DIS
LIN {X 35.32, Y 228.99, Z 0.00, A 0, B 0, C 0} C_DIS
LIN {X 35.24, Y 228.69, Z 0.00, A 0, B 0, C 0} C_DIS
LIN {X 35.15, Y 228.39, Z 0.00, A 0, B 0, C 0} C_DIS
LIN {X 35.07, Y 228.09, Z 0.00, A 0, B 0, C 0} C_DIS
LIN {X 35.02, Y 227.77, Z 0.00, A 0, B 0, C 0} C_DIS
LIN {X 34.97, Y 227.45, Z 0.00, A 0, B 0, C 0} C_DIS
LIN {X 34.91, Y 227.13, Z 0.00, A 0, B 0, C 0} C_DIS
LIN {X 34.83, Y 226.83, Z 0.00, A 0, B 0, C 0} C_DIS
LIN {X 34.75, Y 226.53, Z 0.00, A 0, B 0, C 0} C_DIS
LIN {X 34.67, Y 226.22, Z 0.00, A 0, B 0, C 0} C_DIS
LIN {X 34.60, Y 225.91, Z 0.00, A 0, B 0, C 0} C_DIS
LIN {X 34.53, Y 225.60, Z 0.00, A 0, B 0, C 0} C_DIS
LIN {X 34.46, Y 225.30, Z 0.00, A 0, B 0, C 0} C_DIS
LIN {X 34.35, Y 225.01, Z 0.00, A 0, B 0, C 0} C_DIS
LIN {X 34.24, Y 224.73, Z 0.00, A 0, B 0, C 0} C_DIS
LIN {X 34.14, Y 224.44, Z 0.00, A 0, B 0, C 0} C_DIS
LIN {X 34.08, Y 224.13, Z 0.00, A 0, B 0, C 0} C_DIS
LIN {X 34.03, Y 223.80, Z 0.00, A 0, B 0, C 0} C_DIS
LIN {X 33.99, Y 223.48, Z 0.00, A 0, B 0, C 0} C_DIS
LIN {X 33.94, Y 223.16, Z 0.00, A 0, B 0, C 0} C_DIS
LIN {X 33.88, Y 222.85, Z 0.00, A 0, B 0, C 0} C_DIS
LIN {X 33.83, Y 222.53, Z 0.00, A 0, B 0, C 0} C_DIS
LIN {X 33.77, Y 222.21, Z 0.00, A 0, B 0, C 0} C_DIS
LIN {X 33.72, Y 221.90, Z 0.00, A 0, B 0, C 0} C_DIS
LIN {X 33.66, Y 221.58, Z 0.00, A 0, B 0, C 0} C_DIS
LIN {X 33.61, Y 221.26, Z 0.00, A 0, B 0, C 0} C_DIS
LIN {X 33.57, Y 220.94, Z 0.00, A 0, B 0, C 0} C_DIS
LIN {X 33.53, Y 220.62, Z 0.00, A 0, B 0, C 0} C_DIS
LIN {X 33.50, Y 220.29, Z 0.00, A 0, B 0, C 0} C_DIS
LIN {X 33.47, Y 219.97, Z 0.00, A 0, B 0, C 0} C_DIS
LIN {X 33.44, Y 219.65, Z 0.00, A 0, B 0, C 0} C_DIS
LIN {X 33.41, Y 219.32, Z 0.00, A 0, B 0, C 0} C_DIS
LIN {X 33.36, Y 219.00, Z 0.00, A 0, B 0, C 0} C_DIS
LIN {X 33.30, Y 218.69, Z 0.00, A 0, B 0, C 0} C_DIS
LIN {X 33.24, Y 218.37, Z 0.00, A 0, B 0, C 0} C_DIS
LIN {X 33.18, Y 218.05, Z 0.00, A 0, B 0, C 0} C_DIS
LIN {X 33.13, Y 217.73, Z 0.00, A 0, B 0, C 0} C_DIS
LIN {X 33.10, Y 217.41, Z 0.00, A 0, B 0, C 0} C_DIS
LIN {X 33.07, Y 217.09, Z 0.00, A 0, B 0, C 0} C_DIS
LIN {X 33.06, Y 216.76, Z 0.00, A 0, B 0, C 0} C_DIS
LIN {X 33.05, Y 216.44, Z 0.00, A 0, B 0, C 0} C_DIS
LIN {X 33.04, Y 216.11, Z 0.00, A 0, B 0, C 0} C_DIS
LIN {X 33.02, Y 215.78, Z 0.00, A 0, B 0, C 0} C_DIS
LIN {X 32.99, Y 215.46, Z 0.00, A 0, B 0, C 0} C_DIS
LIN {X 32.94, Y 215.14, Z 0.00, A 0, B 0, C 0} C_DIS
LIN {X 32.88, Y 214.82, Z 0.00, A 0, B 0, C 0} C_DIS
LIN {X 32.82, Y 214.51, Z 0.00, A 0, B 0, C 0} C_DIS
LIN {X 32.76, Y 214.19, Z 0.00, A 0, B 0, C 0} C_DIS
LIN {X 32.71, Y 213.87, Z 0.00, A 0, B 0, C 0} C_DIS
LIN {X 32.67, Y 213.55, Z 0.00, A 0, B 0, C 0} C_DIS
LIN {X 32.64, Y 213.23, Z 0.00, A 0, B 0, C 0} C_DIS
LIN {X 32.62, Y 212.90, Z 0.00, A 0, B 0, C 0} C_DIS
LIN {X 32.62, Y 212.57, Z 0.00, A 0, B 0, C 0} C_DIS
LIN {X 32.62, Y 212.25, Z 0.00, A 0, B 0, C 0} C_DIS
LIN {X 32.62, Y 211.92, Z 0.00, A 0, B 0, C 0} C_DIS
LIN {X 32.62, Y 211.59, Z 0.00, A 0, B 0, C 0} C_DIS
LIN {X 32.62, Y 211.26, Z 0.00, A 0, B 0, C 0} C_DIS
LIN {X 32.62, Y 210.94, Z 0.00, A 0, B 0, C 0} C_DIS
LIN {X 32.62, Y 210.61, Z 0.00, A 0, B 0, C 0} C_DIS
LIN {X 32.62, Y 210.28, Z 0.00, A 0, B 0, C 0} C_DIS
LIN {X 32.62, Y 209.95, Z 0.00, A 0, B 0, C 0} C_DIS
LIN {X 32.62, Y 209.62, Z 0.00, A 0, B 0, C 0} C_DIS
LIN {X 32.62, Y 209.30, Z 0.00, A 0, B 0, C 0} C_DIS
LIN {X 32.62, Y 208.97, Z 0.00, A 0, B 0, C 0} C_DIS
LIN {X 32.62, Y 208.64, Z 0.00, A 0, B 0, C 0} C_DIS
LIN {X 32.62, Y 208.32, Z 0.00, A 0, B 0, C 0} C_DIS
LIN {X 32.63, Y 207.99, Z 0.00, A 0, B 0, C 0} C_DIS
LIN {X 32.63, Y 207.66, Z 0.00, A 0, B 0, C 0} C_DIS
LIN {X 32.62, Y 207.33, Z 0.00, A 0, B 0, C 0} C_DIS
LIN {X 32.62, Y 207.00, Z 0.00, A 0, B 0, C 0} C_DIS
LIN {X 32.61, Y 206.67, Z 0.00, A 0, B 0, C 0} C_DIS
LIN {X 32.61, Y 206.35, Z 0.00, A 0, B 0, C 0} C_DIS
LIN {X 32.61, Y 206.02, Z 0.00, A 0, B 0, C 0} C_DIS
LIN {X 32.62, Y 205.69, Z 0.00, A 0, B 0, C 0} C_DIS
LIN {X 32.64, Y 205.37, Z 0.00, A 0, B 0, C 0} C_DIS
LIN {X 32.67, Y 205.04, Z 0.00, A 0, B 0, C 0} C_DIS
LIN {X 32.72, Y 204.72, Z 0.00, A 0, B 0, C 0} C_DIS
LIN {X 32.77, Y 204.41, Z 0.00, A 0, B 0, C 0} C_DIS
LIN {X 32.83, Y 204.09, Z 0.00, A 0, B 0, C 0} C_DIS
LIN {X 32.88, Y 203.77, Z 0.00, A 0, B 0, C 0} C_DIS
LIN {X 32.94, Y 203.45, Z 0.00, A 0, B 0, C 0} C_DIS
LIN {X 32.98, Y 203.13, Z 0.00, A 0, B 0, C 0} C_DIS
LIN {X 33.02, Y 202.81, Z 0.00, A 0, B 0, C 0} C_DIS
LIN {X 33.04, Y 202.49, Z 0.00, A 0, B 0, C 0} C_DIS
LIN {X 33.06, Y 202.16, Z 0.00, A 0, B 0, C 0} C_DIS
LIN {X 33.07, Y 201.83, Z 0.00, A 0, B 0, C 0} C_DIS
LIN {X 33.08, Y 201.51, Z 0.00, A 0, B 0, C 0} C_DIS
LIN {X 33.10, Y 201.18, Z 0.00, A 0, B 0, C 0} C_DIS
LIN {X 33.14, Y 200.86, Z 0.00, A 0, B 0, C 0} C_DIS
LIN {X 33.19, Y 200.54, Z 0.00, A 0, B 0, C 0} C_DIS
LIN {X 33.24, Y 200.22, Z 0.00, A 0, B 0, C 0} C_DIS
LIN {X 33.30, Y 199.91, Z 0.00, A 0, B 0, C 0} C_DIS
LIN {X 33.35, Y 199.59, Z 0.00, A 0, B 0, C 0} C_DIS
LIN {X 33.41, Y 199.27, Z 0.00, A 0, B 0, C 0} C_DIS
LIN {X 33.46, Y 198.95, Z 0.00, A 0, B 0, C 0} C_DIS
LIN {X 33.52, Y 198.64, Z 0.00, A 0, B 0, C 0} C_DIS
LIN {X 33.57, Y 198.32, Z 0.00, A 0, B 0, C 0} C_DIS
LIN {X 33.62, Y 198.00, Z 0.00, A 0, B 0, C 0} C_DIS
LIN {X 33.68, Y 197.68, Z 0.00, A 0, B 0, C 0} C_DIS
LIN {X 33.73, Y 197.37, Z 0.00, A 0, B 0, C 0} C_DIS
LIN {X 33.78, Y 197.05, Z 0.00, A 0, B 0, C 0} C_DIS
LIN {X 33.83, Y 196.73, Z 0.00, A 0, B 0, C 0} C_DIS
LIN {X 33.88, Y 196.41, Z 0.00, A 0, B 0, C 0} C_DIS
LIN {X 33.93, Y 196.09, Z 0.00, A 0, B 0, C 0} C_DIS
LIN {X 33.98, Y 195.77, Z 0.00, A 0, B 0, C 0} C_DIS
LIN {X 34.03, Y 195.45, Z 0.00, A 0, B 0, C 0} C_DIS
LIN {X 34.09, Y 195.14, Z 0.00, A 0, B 0, C 0} C_DIS
LIN {X 34.14, Y 194.82, Z 0.00, A 0, B 0, C 0} C_DIS
LIN {X 34.20, Y 194.51, Z 0.00, A 0, B 0, C 0} C_DIS
LIN {X 34.28, Y 194.20, Z 0.00, A 0, B 0, C 0} C_DIS
LIN {X 34.36, Y 193.90, Z 0.00, A 0, B 0, C 0} C_DIS
LIN {X 34.44, Y 193.59, Z 0.00, A 0, B 0, C 0} C_DIS
LIN {X 34.50, Y 193.28, Z 0.00, A 0, B 0, C 0} C_DIS
LIN {X 34.57, Y 192.97, Z 0.00, A 0, B 0, C 0} C_DIS
LIN {X 34.64, Y 192.66, Z 0.00, A 0, B 0, C 0} C_DIS
LIN {X 34.75, Y 192.37, Z 0.00, A 0, B 0, C 0} C_DIS
LIN {X 34.86, Y 192.10, Z 0.00, A 0, B 0, C 0} C_DIS
LIN {X 34.95, Y 191.80, Z 0.00, A 0, B 0, C 0} C_DIS
LIN {X 35.03, Y 191.49, Z 0.00, A 0, B 0, C 0} C_DIS
LIN {X 35.09, Y 191.18, Z 0.00, A 0, B 0, C 0} C_DIS
LIN {X 35.15, Y 190.87, Z 0.00, A 0, B 0, C 0} C_DIS
LIN {X 35.23, Y 190.56, Z 0.00, A 0, B 0, C 0} C_DIS
LIN {X 35.32, Y 190.26, Z 0.00, A 0, B 0, C 0} C_DIS
LIN {X 35.39, Y 189.96, Z 0.00, A 0, B 0, C 0} C_DIS
LIN {X 35.45, Y 189.64, Z 0.00, A 0, B 0, C 0} C_DIS
LIN {X 35.52, Y 189.33, Z 0.00, A 0, B 0, C 0} C_DIS
LIN {X 35.63, Y 189.05, Z 0.00, A 0, B 0, C 0} C_DIS
LIN {X 35.75, Y 188.77, Z 0.00, A 0, B 0, C 0} C_DIS
LIN {X 35.84, Y 188.47, Z 0.00, A 0, B 0, C 0} C_DIS
LIN {X 35.92, Y 188.17, Z 0.00, A 0, B 0, C 0} C_DIS
LIN {X 36.01, Y 187.88, Z 0.00, A 0, B 0, C 0} C_DIS
LIN {X 36.13, Y 187.60, Z 0.00, A 0, B 0, C 0} C_DIS
LIN {X 36.23, Y 187.31, Z 0.00, A 0, B 0, C 0} C_DIS
LIN {X 36.31, Y 187.01, Z 0.00, A 0, B 0, C 0} C_DIS
LIN {X 36.40, Y 186.71, Z 0.00, A 0, B 0, C 0} C_DIS
LIN {X 36.51, Y 186.42, Z 0.00, A 0, B 0, C 0} C_DIS
LIN {X 36.62, Y 186.14, Z 0.00, A 0, B 0, C 0} C_DIS
LIN {X 36.71, Y 185.85, Z 0.00, A 0, B 0, C 0} C_DIS
LIN {X 36.79, Y 185.54, Z 0.00, A 0, B 0, C 0} C_DIS
LIN {X 36.89, Y 185.25, Z 0.00, A 0, B 0, C 0} C_DIS
LIN {X 37.00, Y 184.97, Z 0.00, A 0, B 0, C 0} C_DIS
LIN {X 37.12, Y 184.70, Z 0.00, A 0, B 0, C 0} C_DIS
LIN {X 37.24, Y 184.43, Z 0.00, A 0, B 0, C 0} C_DIS
LIN {X 37.37, Y 184.16, Z 0.00, A 0, B 0, C 0} C_DIS
LIN {X 37.49, Y 183.88, Z 0.00, A 0, B 0, C 0} C_DIS
LIN {X 37.61, Y 183.61, Z 0.00, A 0, B 0, C 0} C_DIS
LIN {X 37.73, Y 183.34, Z 0.00, A 0, B 0, C 0} C_DIS
LIN {X 37.85, Y 183.06, Z 0.00, A 0, B 0, C 0} C_DIS
LIN {X 37.97, Y 182.79, Z 0.00, A 0, B 0, C 0} C_DIS
LIN {X 38.09, Y 182.52, Z 0.00, A 0, B 0, C 0} C_DIS
LIN {X 38.21, Y 182.24, Z 0.00, A 0, B 0, C 0} C_DIS
LIN {X 38.33, Y 181.97, Z 0.00, A 0, B 0, C 0} C_DIS
LIN {X 38.45, Y 181.70, Z 0.00, A 0, B 0, C 0} C_DIS
LIN {X 38.57, Y 181.43, Z 0.00, A 0, B 0, C 0} C_DIS
LIN {X 38.69, Y 181.16, Z 0.00, A 0, B 0, C 0} C_DIS
LIN {X 38.81, Y 180.88, Z 0.00, A 0, B 0, C 0} C_DIS
LIN {X 38.93, Y 180.60, Z 0.00, A 0, B 0, C 0} C_DIS
LIN {X 39.05, Y 180.33, Z 0.00, A 0, B 0, C 0} C_DIS
LIN {X 39.19, Y 180.08, Z 0.00, A 0, B 0, C 0} C_DIS
LIN {X 39.34, Y 179.85, Z 0.00, A 0, B 0, C 0} C_DIS
LIN {X 39.49, Y 179.62, Z 0.00, A 0, B 0, C 0} C_DIS
LIN {X 39.63, Y 179.36, Z 0.00, A 0, B 0, C 0} C_DIS
LIN {X 39.75, Y 179.09, Z 0.00, A 0, B 0, C 0} C_DIS
LIN {X 39.87, Y 178.82, Z 0.00, A 0, B 0, C 0} C_DIS
LIN {X 39.99, Y 178.54, Z 0.00, A 0, B 0, C 0} C_DIS
LIN {X 40.11, Y 178.27, Z 0.00, A 0, B 0, C 0} C_DIS
LIN {X 40.23, Y 178.00, Z 0.00, A 0, B 0, C 0} C_DIS
LIN {X 40.35, Y 177.73, Z 0.00, A 0, B 0, C 0} C_DIS
LIN {X 40.49, Y 177.47, Z 0.00, A 0, B 0, C 0} C_DIS
LIN {X 40.63, Y 177.23, Z 0.00, A 0, B 0, C 0} C_DIS
LIN {X 40.79, Y 177.00, Z 0.00, A 0, B 0, C 0} C_DIS
LIN {X 40.94, Y 176.77, Z 0.00, A 0, B 0, C 0} C_DIS
LIN {X 41.10, Y 176.54, Z 0.00, A 0, B 0, C 0} C_DIS
LIN {X 41.25, Y 176.31, Z 0.00, A 0, B 0, C 0} C_DIS
LIN {X 41.41, Y 176.08, Z 0.00, A 0, B 0, C 0} C_DIS
LIN {X 41.56, Y 175.85, Z 0.00, A 0, B 0, C 0} C_DIS
LIN {X 41.72, Y 175.62, Z 0.00, A 0, B 0, C 0} C_DIS
LIN {X 41.87, Y 175.39, Z 0.00, A 0, B 0, C 0} C_DIS
LIN {X 42.02, Y 175.15, Z 0.00, A 0, B 0, C 0} C_DIS
LIN {X 42.18, Y 174.92, Z 0.00, A 0, B 0, C 0} C_DIS
LIN {X 42.33, Y 174.69, Z 0.00, A 0, B 0, C 0} C_DIS
LIN {X 42.48, Y 174.46, Z 0.00, A 0, B 0, C 0} C_DIS
LIN {X 42.64, Y 174.22, Z 0.00, A 0, B 0, C 0} C_DIS
LIN {X 42.79, Y 173.99, Z 0.00, A 0, B 0, C 0} C_DIS
LIN {X 42.94, Y 173.76, Z 0.00, A 0, B 0, C 0} C_DIS
LIN {X 43.10, Y 173.52, Z 0.00, A 0, B 0, C 0} C_DIS
LIN {X 43.25, Y 173.29, Z 0.00, A 0, B 0, C 0} C_DIS
LIN {X 43.41, Y 173.06, Z 0.00, A 0, B 0, C 0} C_DIS
LIN {X 43.56, Y 172.84, Z 0.00, A 0, B 0, C 0} C_DIS
LIN {X 43.73, Y 172.63, Z 0.00, A 0, B 0, C 0} C_DIS
LIN {X 43.90, Y 172.42, Z 0.00, A 0, B 0, C 0} C_DIS
LIN {X 44.07, Y 172.23, Z 0.00, A 0, B 0, C 0} C_DIS
LIN {X 44.26, Y 172.06, Z 0.00, A 0, B 0, C 0} C_DIS
LIN {X 44.44, Y 171.89, Z 0.00, A 0, B 0, C 0} C_DIS
LIN {X 44.63, Y 171.71, Z 0.00, A 0, B 0, C 0} C_DIS
LIN {X 44.81, Y 171.53, Z 0.00, A 0, B 0, C 0} C_DIS
LIN {X 44.98, Y 171.33, Z 0.00, A 0, B 0, C 0} C_DIS
LIN {X 45.14, Y 171.11, Z 0.00, A 0, B 0, C 0} C_DIS
LIN {X 45.29, Y 170.88, Z 0.00, A 0, B 0, C 0} C_DIS
LIN {X 45.44, Y 170.64, Z 0.00, A 0, B 0, C 0} C_DIS
LIN {X 45.60, Y 170.40, Z 0.00, A 0, B 0, C 0} C_DIS
LIN {X 45.76, Y 170.18, Z 0.00, A 0, B 0, C 0} C_DIS
LIN {X 45.92, Y 169.98, Z 0.00, A 0, B 0, C 0} C_DIS
LIN {X 46.10, Y 169.79, Z 0.00, A 0, B 0, C 0} C_DIS
LIN {X 46.28, Y 169.60, Z 0.00, A 0, B 0, C 0} C_DIS
LIN {X 46.46, Y 169.41, Z 0.00, A 0, B 0, C 0} C_DIS
LIN {X 46.64, Y 169.23, Z 0.00, A 0, B 0, C 0} C_DIS
LIN {X 46.82, Y 169.05, Z 0.00, A 0, B 0, C 0} C_DIS
LIN {X 47.00, Y 168.88, Z 0.00, A 0, B 0, C 0} C_DIS
LIN {X 47.19, Y 168.70, Z 0.00, A 0, B 0, C 0} C_DIS
LIN {X 47.37, Y 168.52, Z 0.00, A 0, B 0, C 0} C_DIS
LIN {X 47.55, Y 168.33, Z 0.00, A 0, B 0, C 0} C_DIS
LIN {X 47.73, Y 168.15, Z 0.00, A 0, B 0, C 0} C_DIS
LIN {X 47.91, Y 167.97, Z 0.00, A 0, B 0, C 0} C_DIS
LIN {X 48.09, Y 167.78, Z 0.00, A 0, B 0, C 0} C_DIS
LIN {X 48.27, Y 167.60, Z 0.00, A 0, B 0, C 0} C_DIS
LIN {X 48.45, Y 167.42, Z 0.00, A 0, B 0, C 0} C_DIS
LIN {X 48.63, Y 167.24, Z 0.00, A 0, B 0, C 0} C_DIS
LIN {X 48.81, Y 167.06, Z 0.00, A 0, B 0, C 0} C_DIS
LIN {X 48.99, Y 166.88, Z 0.00, A 0, B 0, C 0} C_DIS
LIN {X 49.17, Y 166.70, Z 0.00, A 0, B 0, C 0} C_DIS
LIN {X 49.36, Y 166.52, Z 0.00, A 0, B 0, C 0} C_DIS
LIN {X 49.54, Y 166.33, Z 0.00, A 0, B 0, C 0} C_DIS
LIN {X 49.72, Y 166.15, Z 0.00, A 0, B 0, C 0} C_DIS
LIN {X 49.90, Y 165.97, Z 0.00, A 0, B 0, C 0} C_DIS
LIN {X 50.08, Y 165.79, Z 0.00, A 0, B 0, C 0} C_DIS
LIN {X 50.26, Y 165.60, Z 0.00, A 0, B 0, C 0} C_DIS
LIN {X 50.44, Y 165.42, Z 0.00, A 0, B 0, C 0} C_DIS
LIN {X 50.62, Y 165.24, Z 0.00, A 0, B 0, C 0} C_DIS
LIN {X 50.80, Y 165.06, Z 0.00, A 0, B 0, C 0} C_DIS
LIN {X 50.98, Y 164.87, Z 0.00, A 0, B 0, C 0} C_DIS
LIN {X 51.16, Y 164.69, Z 0.00, A 0, B 0, C 0} C_DIS
LIN {X 51.34, Y 164.51, Z 0.00, A 0, B 0, C 0} C_DIS
LIN {X 51.53, Y 164.33, Z 0.00, A 0, B 0, C 0} C_DIS
LIN {X 51.71, Y 164.16, Z 0.00, A 0, B 0, C 0} C_DIS
LIN {X 51.89, Y 163.99, Z 0.00, A 0, B 0, C 0} C_DIS
LIN {X 52.09, Y 163.84, Z 0.00, A 0, B 0, C 0} C_DIS
LIN {X 52.29, Y 163.71, Z 0.00, A 0, B 0, C 0} C_DIS
LIN {X 52.49, Y 163.58, Z 0.00, A 0, B 0, C 0} C_DIS
LIN {X 52.67, Y 163.42, Z 0.00, A 0, B 0, C 0} C_DIS
LIN {X 52.85, Y 163.23, Z 0.00, A 0, B 0, C 0} C_DIS
LIN {X 53.03, Y 163.03, Z 0.00, A 0, B 0, C 0} C_DIS
LIN {X 53.21, Y 162.85, Z 0.00, A 0, B 0, C 0} C_DIS
LIN {X 53.39, Y 162.67, Z 0.00, A 0, B 0, C 0} C_DIS
LIN {X 53.57, Y 162.49, Z 0.00, A 0, B 0, C 0} C_DIS
LIN {X 53.76, Y 162.32, Z 0.00, A 0, B 0, C 0} C_DIS
LIN {X 53.94, Y 162.14, Z 0.00, A 0, B 0, C 0} C_DIS
LIN {X 54.12, Y 161.96, Z 0.00, A 0, B 0, C 0} C_DIS
LIN {X 54.30, Y 161.77, Z 0.00, A 0, B 0, C 0} C_DIS
LIN {X 54.48, Y 161.58, Z 0.00, A 0, B 0, C 0} C_DIS
LIN {X 54.65, Y 161.39, Z 0.00, A 0, B 0, C 0} C_DIS
LIN {X 54.83, Y 161.21, Z 0.00, A 0, B 0, C 0} C_DIS
LIN {X 55.02, Y 161.03, Z 0.00, A 0, B 0, C 0} C_DIS
LIN {X 55.20, Y 160.86, Z 0.00, A 0, B 0, C 0} C_DIS
LIN {X 55.39, Y 160.71, Z 0.00, A 0, B 0, C 0} C_DIS
LIN {X 55.59, Y 160.57, Z 0.00, A 0, B 0, C 0} C_DIS
LIN {X 55.79, Y 160.43, Z 0.00, A 0, B 0, C 0} C_DIS
LIN {X 55.98, Y 160.28, Z 0.00, A 0, B 0, C 0} C_DIS
LIN {X 56.16, Y 160.11, Z 0.00, A 0, B 0, C 0} C_DIS
LIN {X 56.35, Y 159.93, Z 0.00, A 0, B 0, C 0} C_DIS
LIN {X 56.53, Y 159.75, Z 0.00, A 0, B 0, C 0} C_DIS
LIN {X 56.71, Y 159.57, Z 0.00, A 0, B 0, C 0} C_DIS
LIN {X 56.89, Y 159.38, Z 0.00, A 0, B 0, C 0} C_DIS
LIN {X 57.07, Y 159.20, Z 0.00, A 0, B 0, C 0} C_DIS
LIN {X 57.25, Y 159.02, Z 0.00, A 0, B 0, C 0} C_DIS
LIN {X 57.43, Y 158.83, Z 0.00, A 0, B 0, C 0} C_DIS
LIN {X 57.61, Y 158.65, Z 0.00, A 0, B 0, C 0} C_DIS
LIN {X 57.79, Y 158.47, Z 0.00, A 0, B 0, C 0} C_DIS
LIN {X 57.97, Y 158.29, Z 0.00, A 0, B 0, C 0} C_DIS
LIN {X 58.15, Y 158.11, Z 0.00, A 0, B 0, C 0} C_DIS
LIN {X 58.34, Y 157.93, Z 0.00, A 0, B 0, C 0} C_DIS
LIN {X 58.52, Y 157.75, Z 0.00, A 0, B 0, C 0} C_DIS
LIN {X 58.70, Y 157.57, Z 0.00, A 0, B 0, C 0} C_DIS
LIN {X 58.89, Y 157.41, Z 0.00, A 0, B 0, C 0} C_DIS
LIN {X 59.08, Y 157.26, Z 0.00, A 0, B 0, C 0} C_DIS
LIN {X 59.28, Y 157.14, Z 0.00, A 0, B 0, C 0} C_DIS
LIN {X 59.48, Y 157.00, Z 0.00, A 0, B 0, C 0} C_DIS
LIN {X 59.66, Y 156.83, Z 0.00, A 0, B 0, C 0} C_DIS
LIN {X 59.84, Y 156.63, Z 0.00, A 0, B 0, C 0} C_DIS
LIN {X 60.02, Y 156.45, Z 0.00, A 0, B 0, C 0} C_DIS
LIN {X 60.20, Y 156.27, Z 0.00, A 0, B 0, C 0} C_DIS
LIN {X 60.38, Y 156.09, Z 0.00, A 0, B 0, C 0} C_DIS
LIN {X 60.56, Y 155.91, Z 0.00, A 0, B 0, C 0} C_DIS
LIN {X 60.74, Y 155.72, Z 0.00, A 0, B 0, C 0} C_DIS
LIN {X 60.92, Y 155.54, Z 0.00, A 0, B 0, C 0} C_DIS
LIN {X 61.12, Y 155.39, Z 0.00, A 0, B 0, C 0} C_DIS
LIN {X 61.32, Y 155.27, Z 0.00, A 0, B 0, C 0} C_DIS
LIN {X 61.52, Y 155.14, Z 0.00, A 0, B 0, C 0} C_DIS
LIN {X 61.71, Y 154.98, Z 0.00, A 0, B 0, C 0} C_DIS
LIN {X 61.89, Y 154.79, Z 0.00, A 0, B 0, C 0} C_DIS
LIN {X 62.07, Y 154.61, Z 0.00, A 0, B 0, C 0} C_DIS
LIN {X 62.25, Y 154.44, Z 0.00, A 0, B 0, C 0} C_DIS
LIN {X 62.43, Y 154.25, Z 0.00, A 0, B 0, C 0} C_DIS
LIN {X 62.61, Y 154.06, Z 0.00, A 0, B 0, C 0} C_DIS
LIN {X 62.79, Y 153.87, Z 0.00, A 0, B 0, C 0} C_DIS
LIN {X 62.97, Y 153.70, Z 0.00, A 0, B 0, C 0} C_DIS
LIN {X 63.16, Y 153.54, Z 0.00, A 0, B 0, C 0} C_DIS
LIN {X 63.35, Y 153.40, Z 0.00, A 0, B 0, C 0} C_DIS
LIN {X 63.55, Y 153.26, Z 0.00, A 0, B 0, C 0} C_DIS
LIN {X 63.75, Y 153.12, Z 0.00, A 0, B 0, C 0} C_DIS
LIN {X 63.94, Y 152.96, Z 0.00, A 0, B 0, C 0} C_DIS
LIN {X 64.12, Y 152.79, Z 0.00, A 0, B 0, C 0} C_DIS
LIN {X 64.30, Y 152.59, Z 0.00, A 0, B 0, C 0} C_DIS
LIN {X 64.48, Y 152.41, Z 0.00, A 0, B 0, C 0} C_DIS
LIN {X 64.66, Y 152.23, Z 0.00, A 0, B 0, C 0} C_DIS
LIN {X 64.84, Y 152.05, Z 0.00, A 0, B 0, C 0} C_DIS
LIN {X 65.02, Y 151.86, Z 0.00, A 0, B 0, C 0} C_DIS
LIN {X 65.20, Y 151.69, Z 0.00, A 0, B 0, C 0} C_DIS
LIN {X 65.39, Y 151.52, Z 0.00, A 0, B 0, C 0} C_DIS
LIN {X 65.59, Y 151.38, Z 0.00, A 0, B 0, C 0} C_DIS
LIN {X 65.78, Y 151.25, Z 0.00, A 0, B 0, C 0} C_DIS
LIN {X 65.98, Y 151.10, Z 0.00, A 0, B 0, C 0} C_DIS
LIN {X 66.17, Y 150.94, Z 0.00, A 0, B 0, C 0} C_DIS
LIN {X 66.35, Y 150.77, Z 0.00, A 0, B 0, C 0} C_DIS
LIN {X 66.53, Y 150.58, Z 0.00, A 0, B 0, C 0} C_DIS
LIN {X 66.71, Y 150.39, Z 0.00, A 0, B 0, C 0} C_DIS
LIN {X 66.89, Y 150.20, Z 0.00, A 0, B 0, C 0} C_DIS
LIN {X 67.06, Y 150.01, Z 0.00, A 0, B 0, C 0} C_DIS
LIN {X 67.25, Y 149.83, Z 0.00, A 0, B 0, C 0} C_DIS
LIN {X 67.43, Y 149.67, Z 0.00, A 0, B 0, C 0} C_DIS
LIN {X 67.62, Y 149.52, Z 0.00, A 0, B 0, C 0} C_DIS
LIN {X 67.82, Y 149.38, Z 0.00, A 0, B 0, C 0} C_DIS
LIN {X 68.02, Y 149.25, Z 0.00, A 0, B 0, C 0} C_DIS
LIN {X 68.21, Y 149.10, Z 0.00, A 0, B 0, C 0} C_DIS
LIN {X 68.40, Y 148.92, Z 0.00, A 0, B 0, C 0} C_DIS
LIN {X 68.58, Y 148.74, Z 0.00, A 0, B 0, C 0} C_DIS
LIN {X 68.75, Y 148.55, Z 0.00, A 0, B 0, C 0} C_DIS
LIN {X 68.93, Y 148.36, Z 0.00, A 0, B 0, C 0} C_DIS
LIN {X 69.12, Y 148.18, Z 0.00, A 0, B 0, C 0} C_DIS
LIN {X 69.30, Y 148.00, Z 0.00, A 0, B 0, C 0} C_DIS
LIN {X 69.48, Y 147.82, Z 0.00, A 0, B 0, C 0} C_DIS
LIN {X 69.66, Y 147.64, Z 0.00, A 0, B 0, C 0} C_DIS
LIN {X 69.86, Y 147.51, Z 0.00, A 0, B 0, C 0} C_DIS
LIN {X 70.06, Y 147.39, Z 0.00, A 0, B 0, C 0} C_DIS
LIN {X 70.25, Y 147.24, Z 0.00, A 0, B 0, C 0} C_DIS
LIN {X 70.44, Y 147.07, Z 0.00, A 0, B 0, C 0} C_DIS
LIN {X 70.62, Y 146.90, Z 0.00, A 0, B 0, C 0} C_DIS
LIN {X 70.80, Y 146.72, Z 0.00, A 0, B 0, C 0} C_DIS
LIN {X 70.99, Y 146.54, Z 0.00, A 0, B 0, C 0} C_DIS
LIN {X 71.17, Y 146.35, Z 0.00, A 0, B 0, C 0} C_DIS
LIN {X 71.34, Y 146.16, Z 0.00, A 0, B 0, C 0} C_DIS
LIN {X 71.52, Y 145.98, Z 0.00, A 0, B 0, C 0} C_DIS
LIN {X 71.70, Y 145.80, Z 0.00, A 0, B 0, C 0} C_DIS
LIN {X 71.89, Y 145.64, Z 0.00, A 0, B 0, C 0} C_DIS
LIN {X 72.09, Y 145.50, Z 0.00, A 0, B 0, C 0} C_DIS
LIN {X 72.29, Y 145.37, Z 0.00, A 0, B 0, C 0} C_DIS
LIN {X 72.49, Y 145.23, Z 0.00, A 0, B 0, C 0} C_DIS
LIN {X 72.67, Y 145.06, Z 0.00, A 0, B 0, C 0} C_DIS
LIN {X 72.85, Y 144.88, Z 0.00, A 0, B 0, C 0} C_DIS
LIN {X 73.03, Y 144.69, Z 0.00, A 0, B 0, C 0} C_DIS
LIN {X 73.21, Y 144.51, Z 0.00, A 0, B 0, C 0} C_DIS
LIN {X 73.39, Y 144.33, Z 0.00, A 0, B 0, C 0} C_DIS
LIN {X 73.57, Y 144.15, Z 0.00, A 0, B 0, C 0} C_DIS
LIN {X 73.75, Y 143.96, Z 0.00, A 0, B 0, C 0} C_DIS
LIN {X 73.93, Y 143.78, Z 0.00, A 0, B 0, C 0} C_DIS
LIN {X 74.13, Y 143.62, Z 0.00, A 0, B 0, C 0} C_DIS
LIN {X 74.33, Y 143.50, Z 0.00, A 0, B 0, C 0} C_DIS
LIN {X 74.52, Y 143.37, Z 0.00, A 0, B 0, C 0} C_DIS
LIN {X 74.72, Y 143.21, Z 0.00, A 0, B 0, C 0} C_DIS
LIN {X 74.90, Y 143.04, Z 0.00, A 0, B 0, C 0} C_DIS
LIN {X 75.08, Y 142.86, Z 0.00, A 0, B 0, C 0} C_DIS
LIN {X 75.26, Y 142.67, Z 0.00, A 0, B 0, C 0} C_DIS
LIN {X 75.44, Y 142.49, Z 0.00, A 0, B 0, C 0} C_DIS
LIN {X 75.62, Y 142.30, Z 0.00, A 0, B 0, C 0} C_DIS
LIN {X 75.80, Y 142.12, Z 0.00, A 0, B 0, C 0} C_DIS
LIN {X 75.98, Y 141.94, Z 0.00, A 0, B 0, C 0} C_DIS
LIN {X 76.16, Y 141.76, Z 0.00, A 0, B 0, C 0} C_DIS
LIN {X 76.36, Y 141.62, Z 0.00, A 0, B 0, C 0} C_DIS
LIN {X 76.56, Y 141.50, Z 0.00, A 0, B 0, C 0} C_DIS
LIN {X 76.76, Y 141.36, Z 0.00, A 0, B 0, C 0} C_DIS
LIN {X 76.94, Y 141.19, Z 0.00, A 0, B 0, C 0} C_DIS
LIN {X 77.13, Y 141.02, Z 0.00, A 0, B 0, C 0} C_DIS
LIN {X 77.31, Y 140.84, Z 0.00, A 0, B 0, C 0} C_DIS
LIN {X 77.49, Y 140.65, Z 0.00, A 0, B 0, C 0} C_DIS
LIN {X 77.67, Y 140.47, Z 0.00, A 0, B 0, C 0} C_DIS
LIN {X 77.85, Y 140.28, Z 0.00, A 0, B 0, C 0} C_DIS
LIN {X 78.03, Y 140.10, Z 0.00, A 0, B 0, C 0} C_DIS
LIN {X 78.21, Y 139.92, Z 0.00, A 0, B 0, C 0} C_DIS
LIN {X 78.40, Y 139.76, Z 0.00, A 0, B 0, C 0} C_DIS
LIN {X 78.59, Y 139.62, Z 0.00, A 0, B 0, C 0} C_DIS
LIN {X 78.79, Y 139.48, Z 0.00, A 0, B 0, C 0} C_DIS
LIN {X 78.99, Y 139.34, Z 0.00, A 0, B 0, C 0} C_DIS
LIN {X 79.18, Y 139.18, Z 0.00, A 0, B 0, C 0} C_DIS
LIN {X 79.36, Y 139.01, Z 0.00, A 0, B 0, C 0} C_DIS
LIN {X 79.54, Y 138.82, Z 0.00, A 0, B 0, C 0} C_DIS
LIN {X 79.72, Y 138.63, Z 0.00, A 0, B 0, C 0} C_DIS
LIN {X 79.90, Y 138.44, Z 0.00, A 0, B 0, C 0} C_DIS
LIN {X 80.08, Y 138.25, Z 0.00, A 0, B 0, C 0} C_DIS
LIN {X 80.26, Y 138.07, Z 0.00, A 0, B 0, C 0} C_DIS
LIN {X 80.44, Y 137.90, Z 0.00, A 0, B 0, C 0} C_DIS
LIN {X 80.63, Y 137.75, Z 0.00, A 0, B 0, C 0} C_DIS
LIN {X 80.83, Y 137.61, Z 0.00, A 0, B 0, C 0} C_DIS
LIN {X 81.03, Y 137.48, Z 0.00, A 0, B 0, C 0} C_DIS
LIN {X 81.22, Y 137.33, Z 0.00, A 0, B 0, C 0} C_DIS
LIN {X 81.41, Y 137.16, Z 0.00, A 0, B 0, C 0} C_DIS
LIN {X 81.60, Y 137.02, Z 0.00, A 0, B 0, C 0} C_DIS
LIN {X 81.80, Y 136.89, Z 0.00, A 0, B 0, C 0} C_DIS
LIN {X 82.00, Y 136.75, Z 0.00, A 0, B 0, C 0} C_DIS
LIN {X 82.19, Y 136.60, Z 0.00, A 0, B 0, C 0} C_DIS
LIN {X 82.37, Y 136.41, Z 0.00, A 0, B 0, C 0} C_DIS
LIN {X 82.55, Y 136.22, Z 0.00, A 0, B 0, C 0} C_DIS
LIN {X 82.73, Y 136.04, Z 0.00, A 0, B 0, C 0} C_DIS
LIN {X 82.91, Y 135.86, Z 0.00, A 0, B 0, C 0} C_DIS
LIN {X 83.09, Y 135.68, Z 0.00, A 0, B 0, C 0} C_DIS
LIN {X 83.27, Y 135.50, Z 0.00, A 0, B 0, C 0} C_DIS
LIN {X 83.45, Y 135.31, Z 0.00, A 0, B 0, C 0} C_DIS
LIN {X 83.64, Y 135.14, Z 0.00, A 0, B 0, C 0} C_DIS
LIN {X 83.84, Y 135.02, Z 0.00, A 0, B 0, C 0} C_DIS
LIN {X 84.04, Y 134.89, Z 0.00, A 0, B 0, C 0} C_DIS
LIN {X 84.23, Y 134.74, Z 0.00, A 0, B 0, C 0} C_DIS
LIN {X 84.41, Y 134.57, Z 0.00, A 0, B 0, C 0} C_DIS
LIN {X 84.60, Y 134.39, Z 0.00, A 0, B 0, C 0} C_DIS
LIN {X 84.78, Y 134.21, Z 0.00, A 0, B 0, C 0} C_DIS
LIN {X 84.96, Y 134.02, Z 0.00, A 0, B 0, C 0} C_DIS
LIN {X 85.14, Y 133.84, Z 0.00, A 0, B 0, C 0} C_DIS
LIN {X 85.31, Y 133.65, Z 0.00, A 0, B 0, C 0} C_DIS
LIN {X 85.50, Y 133.47, Z 0.00, A 0, B 0, C 0} C_DIS
LIN {X 85.68, Y 133.30, Z 0.00, A 0, B 0, C 0} C_DIS
LIN {X 85.87, Y 133.14, Z 0.00, A 0, B 0, C 0} C_DIS
LIN {X 86.07, Y 133.00, Z 0.00, A 0, B 0, C 0} C_DIS
LIN {X 86.27, Y 132.87, Z 0.00, A 0, B 0, C 0} C_DIS
LIN {X 86.46, Y 132.73, Z 0.00, A 0, B 0, C 0} C_DIS
LIN {X 86.65, Y 132.57, Z 0.00, A 0, B 0, C 0} C_DIS
LIN {X 86.84, Y 132.42, Z 0.00, A 0, B 0, C 0} C_DIS
LIN {X 87.04, Y 132.28, Z 0.00, A 0, B 0, C 0} C_DIS
LIN {X 87.23, Y 132.14, Z 0.00, A 0, B 0, C 0} C_DIS
LIN {X 87.42, Y 131.98, Z 0.00, A 0, B 0, C 0} C_DIS
LIN {X 87.61, Y 131.81, Z 0.00, A 0, B 0, C 0} C_DIS
LIN {X 87.79, Y 131.63, Z 0.00, A 0, B 0, C 0} C_DIS
LIN {X 87.97, Y 131.44, Z 0.00, A 0, B 0, C 0} C_DIS
LIN {X 88.15, Y 131.25, Z 0.00, A 0, B 0, C 0} C_DIS
LIN {X 88.32, Y 131.06, Z 0.00, A 0, B 0, C 0} C_DIS
LIN {X 88.50, Y 130.88, Z 0.00, A 0, B 0, C 0} C_DIS
LIN {X 88.69, Y 130.70, Z 0.00, A 0, B 0, C 0} C_DIS
LIN {X 88.88, Y 130.55, Z 0.00, A 0, B 0, C 0} C_DIS
LIN {X 89.08, Y 130.42, Z 0.00, A 0, B 0, C 0} C_DIS
LIN {X 89.28, Y 130.28, Z 0.00, A 0, B 0, C 0} C_DIS
LIN {X 89.47, Y 130.13, Z 0.00, A 0, B 0, C 0} C_DIS
LIN {X 89.65, Y 129.97, Z 0.00, A 0, B 0, C 0} C_DIS
LIN {X 89.84, Y 129.79, Z 0.00, A 0, B 0, C 0} C_DIS
LIN {X 90.02, Y 129.60, Z 0.00, A 0, B 0, C 0} C_DIS
LIN {X 90.19, Y 129.41, Z 0.00, A 0, B 0, C 0} C_DIS
LIN {X 90.37, Y 129.22, Z 0.00, A 0, B 0, C 0} C_DIS
LIN {X 90.55, Y 129.04, Z 0.00, A 0, B 0, C 0} C_DIS
LIN {X 90.73, Y 128.86, Z 0.00, A 0, B 0, C 0} C_DIS
LIN {X 90.92, Y 128.69, Z 0.00, A 0, B 0, C 0} C_DIS
LIN {X 91.11, Y 128.55, Z 0.00, A 0, B 0, C 0} C_DIS
LIN {X 91.31, Y 128.41, Z 0.00, A 0, B 0, C 0} C_DIS
LIN {X 91.51, Y 128.27, Z 0.00, A 0, B 0, C 0} C_DIS
LIN {X 91.70, Y 128.11, Z 0.00, A 0, B 0, C 0} C_DIS
LIN {X 91.89, Y 127.95, Z 0.00, A 0, B 0, C 0} C_DIS
LIN {X 92.08, Y 127.82, Z 0.00, A 0, B 0, C 0} C_DIS
LIN {X 92.28, Y 127.69, Z 0.00, A 0, B 0, C 0} C_DIS
LIN {X 92.47, Y 127.54, Z 0.00, A 0, B 0, C 0} C_DIS
LIN {X 92.66, Y 127.37, Z 0.00, A 0, B 0, C 0} C_DIS
LIN {X 92.85, Y 127.20, Z 0.00, A 0, B 0, C 0} C_DIS
LIN {X 93.03, Y 127.02, Z 0.00, A 0, B 0, C 0} C_DIS
LIN {X 93.21, Y 126.83, Z 0.00, A 0, B 0, C 0} C_DIS
LIN {X 93.38, Y 126.64, Z 0.00, A 0, B 0, C 0} C_DIS
LIN {X 93.56, Y 126.45, Z 0.00, A 0, B 0, C 0} C_DIS
LIN {X 93.74, Y 126.27, Z 0.00, A 0, B 0, C 0} C_DIS
LIN {X 93.93, Y 126.10, Z 0.00, A 0, B 0, C 0} C_DIS
LIN {X 94.12, Y 125.95, Z 0.00, A 0, B 0, C 0} C_DIS
LIN {X 94.32, Y 125.81, Z 0.00, A 0, B 0, C 0} C_DIS
LIN {X 94.51, Y 125.67, Z 0.00, A 0, B 0, C 0} C_DIS
LIN {X 94.71, Y 125.52, Z 0.00, A 0, B 0, C 0} C_DIS
LIN {X 94.89, Y 125.36, Z 0.00, A 0, B 0, C 0} C_DIS
LIN {X 95.08, Y 125.18, Z 0.00, A 0, B 0, C 0} C_DIS
LIN {X 95.26, Y 125.00, Z 0.00, A 0, B 0, C 0} C_DIS
LIN {X 95.43, Y 124.81, Z 0.00, A 0, B 0, C 0} C_DIS
LIN {X 95.61, Y 124.62, Z 0.00, A 0, B 0, C 0} C_DIS
LIN {X 95.79, Y 124.43, Z 0.00, A 0, B 0, C 0} C_DIS
LIN {X 95.97, Y 124.25, Z 0.00, A 0, B 0, C 0} C_DIS
LIN {X 96.16, Y 124.08, Z 0.00, A 0, B 0, C 0} C_DIS
LIN {X 96.35, Y 123.94, Z 0.00, A 0, B 0, C 0} C_DIS
LIN {X 96.55, Y 123.81, Z 0.00, A 0, B 0, C 0} C_DIS
LIN {X 96.75, Y 123.67, Z 0.00, A 0, B 0, C 0} C_DIS
LIN {X 96.94, Y 123.51, Z 0.00, A 0, B 0, C 0} C_DIS
LIN {X 97.13, Y 123.35, Z 0.00, A 0, B 0, C 0} C_DIS
LIN {X 97.32, Y 123.21, Z 0.00, A 0, B 0, C 0} C_DIS
LIN {X 97.52, Y 123.08, Z 0.00, A 0, B 0, C 0} C_DIS
LIN {X 97.72, Y 122.93, Z 0.00, A 0, B 0, C 0} C_DIS
LIN {X 97.90, Y 122.77, Z 0.00, A 0, B 0, C 0} C_DIS
LIN {X 98.09, Y 122.60, Z 0.00, A 0, B 0, C 0} C_DIS
LIN {X 98.27, Y 122.41, Z 0.00, A 0, B 0, C 0} C_DIS
LIN {X 98.44, Y 122.22, Z 0.00, A 0, B 0, C 0} C_DIS
LIN {X 98.62, Y 122.03, Z 0.00, A 0, B 0, C 0} C_DIS
LIN {X 98.80, Y 121.84, Z 0.00, A 0, B 0, C 0} C_DIS
LIN {X 98.98, Y 121.66, Z 0.00, A 0, B 0, C 0} C_DIS
LIN {X 99.17, Y 121.50, Z 0.00, A 0, B 0, C 0} C_DIS
LIN {X 99.36, Y 121.35, Z 0.00, A 0, B 0, C 0} C_DIS
LIN {X 99.56, Y 121.21, Z 0.00, A 0, B 0, C 0} C_DIS
LIN {X 99.76, Y 121.08, Z 0.00, A 0, B 0, C 0} C_DIS
LIN {X 99.95, Y 120.92, Z 0.00, A 0, B 0, C 0} C_DIS
LIN {X 100.13, Y 120.75, Z 0.00, A 0, B 0, C 0} C_DIS
LIN {X 100.31, Y 120.57, Z 0.00, A 0, B 0, C 0} C_DIS
LIN {X 100.49, Y 120.38, Z 0.00, A 0, B 0, C 0} C_DIS
LIN {X 100.67, Y 120.20, Z 0.00, A 0, B 0, C 0} C_DIS
LIN {X 100.85, Y 120.02, Z 0.00, A 0, B 0, C 0} C_DIS
LIN {X 101.03, Y 119.83, Z 0.00, A 0, B 0, C 0} C_DIS
LIN {X 101.21, Y 119.65, Z 0.00, A 0, B 0, C 0} C_DIS
LIN {X 101.40, Y 119.47, Z 0.00, A 0, B 0, C 0} C_DIS
LIN {X 101.59, Y 119.33, Z 0.00, A 0, B 0, C 0} C_DIS
LIN {X 101.79, Y 119.21, Z 0.00, A 0, B 0, C 0} C_DIS
LIN {X 101.99, Y 119.07, Z 0.00, A 0, B 0, C 0} C_DIS
LIN {X 102.18, Y 118.90, Z 0.00, A 0, B 0, C 0} C_DIS
LIN {X 102.36, Y 118.74, Z 0.00, A 0, B 0, C 0} C_DIS
LIN {X 102.56, Y 118.61, Z 0.00, A 0, B 0, C 0} C_DIS
LIN {X 102.76, Y 118.48, Z 0.00, A 0, B 0, C 0} C_DIS
LIN {X 102.95, Y 118.33, Z 0.00, A 0, B 0, C 0} C_DIS
LIN {X 103.14, Y 118.16, Z 0.00, A 0, B 0, C 0} C_DIS
LIN {X 103.32, Y 117.99, Z 0.00, A 0, B 0, C 0} C_DIS
LIN {X 103.50, Y 117.80, Z 0.00, A 0, B 0, C 0} C_DIS
LIN {X 103.68, Y 117.61, Z 0.00, A 0, B 0, C 0} C_DIS
LIN {X 103.86, Y 117.42, Z 0.00, A 0, B 0, C 0} C_DIS
LIN {X 104.04, Y 117.23, Z 0.00, A 0, B 0, C 0} C_DIS
LIN {X 104.22, Y 117.06, Z 0.00, A 0, B 0, C 0} C_DIS
LIN {X 104.41, Y 116.90, Z 0.00, A 0, B 0, C 0} C_DIS
LIN {X 104.60, Y 116.75, Z 0.00, A 0, B 0, C 0} C_DIS
LIN {X 104.80, Y 116.60, Z 0.00, A 0, B 0, C 0} C_DIS
LIN {X 104.99, Y 116.46, Z 0.00, A 0, B 0, C 0} C_DIS
LIN {X 105.18, Y 116.31, Z 0.00, A 0, B 0, C 0} C_DIS
LIN {X 105.37, Y 116.15, Z 0.00, A 0, B 0, C 0} C_DIS
LIN {X 105.55, Y 115.97, Z 0.00, A 0, B 0, C 0} C_DIS
LIN {X 105.73, Y 115.78, Z 0.00, A 0, B 0, C 0} C_DIS
LIN {X 105.91, Y 115.59, Z 0.00, A 0, B 0, C 0} C_DIS
LIN {X 106.09, Y 115.40, Z 0.00, A 0, B 0, C 0} C_DIS
LIN {X 106.27, Y 115.22, Z 0.00, A 0, B 0, C 0} C_DIS
LIN {X 106.45, Y 115.04, Z 0.00, A 0, B 0, C 0} C_DIS
LIN {X 106.64, Y 114.88, Z 0.00, A 0, B 0, C 0} C_DIS
LIN {X 106.83, Y 114.73, Z 0.00, A 0, B 0, C 0} C_DIS
LIN {X 107.03, Y 114.59, Z 0.00, A 0, B 0, C 0} C_DIS
LIN {X 107.23, Y 114.46, Z 0.00, A 0, B 0, C 0} C_DIS
LIN {X 107.42, Y 114.30, Z 0.00, A 0, B 0, C 0} C_DIS
LIN {X 107.61, Y 114.14, Z 0.00, A 0, B 0, C 0} C_DIS
LIN {X 107.81, Y 114.01, Z 0.00, A 0, B 0, C 0} C_DIS
LIN {X 108.00, Y 113.88, Z 0.00, A 0, B 0, C 0} C_DIS
